LIN {X 0,Y 364.275,Z 621.196,A -85,B 0,C 180,E1 12256.474,E2 12256.474} C_VEL
LIN {X 0,Y 364.034,Z 587.813,A -85,B 0,C 180,E1 12257.54,E2 12257.54} C_VEL
LIN {X 0,Y 354.056,Z 549.53,A -85,B 0,C 180,E1 12259.048,E2 12259.048} C_VEL
LIN {X 0,Y 353.541,Z 549.53,A -85,B 0,C 180,E1 12266.307,E2 12266.307} C_VEL
LIN {X 0,Y 353.274,Z 549.53,A -85,B 0,C 180,E1 12273.738,E2 12273.738} C_VEL
LIN {X 0,Y 353.185,Z 549.53,A -85,B 0,C 180,E1 12279.866,E2 12279.866} C_VEL
LIN {X 0,Y 353.249,Z 549.563,A -85,B 0,C 180,E1 12286.159,E2 12286.159} C_VEL
LIN {X 0,Y 355.771,Z 555.279,A -85,B 0,C 180,E1 12286.913,E2 12286.913} C_VEL
LIN {X 0,Y 373.351,Z 588.547,A -85,B 0,C 180,E1 12291.308,E2 12291.308} C_VEL
LIN {X 0,Y 385.04,Z 618.639,A -85,B 0,C 180,E1 12294.556,E2 12294.556} C_VEL
LIN {X 0,Y 386.445,Z 626.078,A -85,B 0,C 180,E1 12295.26,E2 12295.26} C_VEL
LIN {X 0,Y 380.974,Z 661.138,A -85,B 0,C 180,E1 12297.839,E2 12297.839} C_VEL
LIN {X 0,Y 374.56,Z 693.358,A -85,B 0,C 180,E1 12301.251,E2 12301.251} C_VEL
LIN {X 0,Y 368.305,Z 721.793,A -85,B 0,C 180,E1 12305.491,E2 12305.491} C_VEL
LIN {X 0,Y 363.131,Z 744.325,A -85,B 0,C 180,E1 12310.113,E2 12310.113} C_VEL
LIN {X 0,Y 359.19,Z 762.864,A -85,B 0,C 180,E1 12315.399,E2 12315.399} C_VEL
LIN {X 0,Y 356.931,Z 776.042,A -85,B 0,C 180,E1 12320.877,E2 12320.877} C_VEL
LIN {X 0,Y 355.982,Z 784.021,A -85,B 0,C 180,E1 12326.354,E2 12326.354} C_VEL
LIN {X 0,Y 355.823,Z 786.74,A -85,B 0,C 180,E1 12330,E2 12330} C_VEL
LIN {X 0,Y 355.614,Z 787.304,A -85,B 0,C 180,E1 12334.869,E2 12334.869} C_VEL
LIN {X 0,Y 356.095,Z 782.784,A -85,B 0,C 180,E1 12340.995,E2 12340.995} C_VEL
LIN {X 0,Y 357.469,Z 773.674,A -85,B 0,C 180,E1 12346.558,E2 12346.558} C_VEL
LIN {X 0,Y 360.3,Z 759.136,A -85,B 0,C 180,E1 12352.147,E2 12352.147} C_VEL
LIN {X 0,Y 365.023,Z 739.076,A -85,B 0,C 180,E1 12357.433,E2 12357.433} C_VEL
LIN {X 0,Y 371.397,Z 713.51,A -85,B 0,C 180,E1 12362.225,E2 12362.225} C_VEL
LIN {X 0,Y 377.949,Z 685.061,A -85,B 0,C 180,E1 12366.085,E2 12366.085} C_VEL
LIN {X 0,Y 384.414,Z 652.218,A -85,B 0,C 180,E1 12369.256,E2 12369.256} C_VEL
LIN {X 0,Y 388.288,Z 623.748,A -85,B 0,C 180,E1 12371.277,E2 12371.277} C_VEL
LIN {X 0,Y 379.667,Z 599.13,A -85,B 0,C 180,E1 12374.088,E2 12374.088} C_VEL
LIN {X 0,Y 362.784,Z 566.88,A -85,B 0,C 180,E1 12378.529,E2 12378.529} C_VEL
LIN {X 0,Y 353.462,Z 550.572,A -85,B 0,C 180,E1 12381.288,E2 12381.288} C_VEL
LIN {X 0,Y 353.384,Z 549.53,A -85,B 0,C 180,E1 12381.533,E2 12381.533} C_VEL
LIN {X 0,Y 353.448,Z 549.53,A -85,B 0,C 180,E1 12389.174,E2 12389.174} C_VEL
LIN {X 0,Y 353.791,Z 549.53,A -85,B 0,C 180,E1 12394.746,E2 12394.746} C_VEL
LIN {X 0,Y 363.12,Z 590.42,A -85,B 0,C 180,E1 12396.235,E2 12396.235} C_VEL
LIN {X 0,Y 362.485,Z 640.026,A -85,B 0,C 180,E1 12397.587,E2 12397.587} C_VEL
LIN {X 0,Y 361.697,Z 666.836,A -85,B 0,C 180,E1 12399.26,E2 12399.26} C_VEL
LIN {X 0,Y 360.494,Z 691.605,A -85,B 0,C 180,E1 12401.855,E2 12401.855} C_VEL
LIN {X 0,Y 359.119,Z 711.774,A -85,B 0,C 180,E1 12405.143,E2 12405.143} C_VEL
LIN {X 0,Y 358.399,Z 725.013,A -85,B 0,C 180,E1 12408.458,E2 12408.458} C_VEL
LIN {X 0,Y 357.994,Z 734.312,A -85,B 0,C 180,E1 12412.298,E2 12412.298} C_VEL
LIN {X 0,Y 358.059,Z 737.826,A -85,B 0,C 180,E1 12415.159,E2 12415.159} C_VEL
LIN {X 0,Y 358.173,Z 738.62,A -85,B 0,C 180,E1 12417.58,E2 12417.58} C_VEL
LIN {X 0,Y 358.909,Z 736.002,A -85,B 0,C 180,E1 12421.199,E2 12421.199} C_VEL
LIN {X 0,Y 360.066,Z 728.623,A -85,B 0,C 180,E1 12424.803,E2 12424.803} C_VEL
LIN {X 0,Y 361.744,Z 715.298,A -85,B 0,C 180,E1 12428.39,E2 12428.39} C_VEL
LIN {X 0,Y 363.572,Z 696.667,A -85,B 0,C 180,E1 12431.517,E2 12431.517} C_VEL
LIN {X 0,Y 365.152,Z 674.086,A -85,B 0,C 180,E1 12433.913,E2 12433.913} C_VEL
LIN {X 0,Y 365.958,Z 647.126,A -85,B 0,C 180,E1 12435.618,E2 12435.618} C_VEL
LIN {X 0,Y 366.369,Z 584.89,A -85,B 0,C 180,E1 12437.501,E2 12437.501} C_VEL
LIN {X 0,Y 357.409,Z 558.523,A -85,B 0,C 180,E1 12439.203,E2 12439.203} C_VEL
LIN {X 0,Y 353.822,Z 549.53,A -85,B 0,C 180,E1 12439.944,E2 12439.944} C_VEL
LIN {X 0,Y 353.455,Z 549.53,A -85,B 0,C 180,E1 12446.277,E2 12446.277} C_VEL
LIN {X 0,Y 353.259,Z 549.53,A -85,B 0,C 180,E1 12454.23,E2 12454.23} C_VEL
LIN {X 0,Y 355.68,Z 555.181,A -85,B 0,C 180,E1 12455.037,E2 12455.037} C_VEL
LIN {X 0,Y 369.418,Z 576.894,A -85,B 0,C 180,E1 12458.683,E2 12458.683} C_VEL
LIN {X 0,Y 385.949,Z 608.362,A -85,B 0,C 180,E1 12462.881,E2 12462.881} C_VEL
LIN {X 0,Y 391.213,Z 623.866,A -85,B 0,C 180,E1 12464.463,E2 12464.463} C_VEL
LIN {X 0,Y 395.036,Z 639.941,A -85,B 0,C 180,E1 12465.933,E2 12465.933} C_VEL
LIN {X 0,Y 388.164,Z 682.729,A -85,B 0,C 180,E1 12468.377,E2 12468.377} C_VEL
LIN {X 0,Y 380.662,Z 723.232,A -85,B 0,C 180,E1 12471.698,E2 12471.698} C_VEL
LIN {X 0,Y 373.751,Z 755.378,A -85,B 0,C 180,E1 12475.4,E2 12475.4} C_VEL
LIN {X 0,Y 367.102,Z 783.844,A -85,B 0,C 180,E1 12479.95,E2 12479.95} C_VEL
LIN {X 0,Y 361.472,Z 808.192,A -85,B 0,C 180,E1 12485.322,E2 12485.322} C_VEL
LIN {X 0,Y 357.553,Z 827.685,A -85,B 0,C 180,E1 12491.408,E2 12491.408} C_VEL
LIN {X 0,Y 355.887,Z 840.326,A -85,B 0,C 180,E1 12497.199,E2 12497.199} C_VEL
LIN {X 0,Y 355.241,Z 848.253,A -85,B 0,C 180,E1 12503.285,E2 12503.285} C_VEL
LIN {X 0,Y 355.256,Z 851.147,A -85,B 0,C 180,E1 12508.729,E2 12508.729} C_VEL
LIN {X 0,Y 352.765,Z 851.098,A -85,B 0,C 180,E1 12510.813,E2 12510.813} C_VEL
LIN {X 0,Y 347.396,Z 849.644,A -85,B 0,C 180,E1 12513.951,E2 12513.951} C_VEL
LIN {X 0,Y 347.31,Z 849.375,A -85,B 0,C 180,E1 12514.316,E2 12514.316} C_VEL
LIN {X 0,Y 347.573,Z 844.231,A -85,B 0,C 180,E1 12520.002,E2 12520.002} C_VEL
LIN {X 0,Y 348.862,Z 833.205,A -85,B 0,C 180,E1 12526.331,E2 12526.331} C_VEL
LIN {X 0,Y 351.743,Z 816.942,A -85,B 0,C 180,E1 12532.382,E2 12532.382} C_VEL
LIN {X 0,Y 356.706,Z 794.96,A -85,B 0,C 180,E1 12538.078,E2 12538.078} C_VEL
LIN {X 0,Y 362.874,Z 769.059,A -85,B 0,C 180,E1 12542.937,E2 12542.937} C_VEL
LIN {X 0,Y 369.91,Z 738.065,A -85,B 0,C 180,E1 12547.128,E2 12547.128} C_VEL
LIN {X 0,Y 377.086,Z 701.811,A -85,B 0,C 180,E1 12550.606,E2 12550.606} C_VEL
LIN {X 0,Y 384.419,Z 658.93,A -85,B 0,C 180,E1 12553.528,E2 12553.528} C_VEL
LIN {X 0,Y 387.166,Z 639.433,A -85,B 0,C 180,E1 12554.558,E2 12554.558} C_VEL
LIN {X 0,Y 379.222,Z 613.621,A -85,B 0,C 180,E1 12557.069,E2 12557.069} C_VEL
LIN {X 0,Y 363.452,Z 581.4,A -85,B 0,C 180,E1 12561.01,E2 12561.01} C_VEL
LIN {X 0,Y 347.32,Z 554.675,A -85,B 0,C 180,E1 12565.104,E2 12565.104} C_VEL
LIN {X 0,Y 345.809,Z 552.078,A -85,B 0,C 180,E1 12565.608,E2 12565.608} C_VEL
LIN {X 0,Y 353.795,Z 566.714,A -85,B 0,C 180,E1 12567.716,E2 12567.716} C_VEL
LIN {X 0,Y 361.627,Z 587.377,A -85,B 0,C 180,E1 12569.616,E2 12569.616} C_VEL
LIN {X 0,Y 362.821,Z 598.343,A -85,B 0,C 180,E1 12570.16,E2 12570.16} C_VEL
LIN {X 0,Y 361.897,Z 640.267,A -85,B 0,C 180,E1 12571.732,E2 12571.732} C_VEL
LIN {X 0,Y 360.473,Z 667.942,A -85,B 0,C 180,E1 12573.669,E2 12573.669} C_VEL
LIN {X 0,Y 358.319,Z 692.777,A -85,B 0,C 180,E1 12576.423,E2 12576.423} C_VEL
LIN {X 0,Y 355.91,Z 713.04,A -85,B 0,C 180,E1 12579.869,E2 12579.869} C_VEL
LIN {X 0,Y 353.542,Z 727.584,A -85,B 0,C 180,E1 12583.724,E2 12583.724} C_VEL
LIN {X 0,Y 351.936,Z 736.22,A -85,B 0,C 180,E1 12587.626,E2 12587.626} C_VEL
LIN {X 0,Y 350.714,Z 740.148,A -85,B 0,C 180,E1 12591.777,E2 12591.777} C_VEL
LIN {X 0,Y 350.188,Z 738.761,A -85,B 0,C 180,E1 12596.3,E2 12596.3} C_VEL
LIN {X 0,Y 350.267,Z 731.975,A -85,B 0,C 180,E1 12600.623,E2 12600.623} C_VEL
LIN {X 0,Y 350.905,Z 719.455,A -85,B 0,C 180,E1 12604.94,E2 12604.94} C_VEL
LIN {X 0,Y 352.138,Z 701.16,A -85,B 0,C 180,E1 12608.942,E2 12608.942} C_VEL
LIN {X 0,Y 353.808,Z 678.257,A -85,B 0,C 180,E1 12612.319,E2 12612.319} C_VEL
LIN {X 0,Y 355.433,Z 652.196,A -85,B 0,C 180,E1 12614.911,E2 12614.911} C_VEL
LIN {X 0,Y 356.666,Z 622.078,A -85,B 0,C 180,E1 12616.775,E2 12616.775} C_VEL
LIN {X 0,Y 356.435,Z 589.165,A -85,B 0,C 180,E1 12617.849,E2 12617.849} C_VEL
LIN {X 0,Y 346.097,Z 549.53,A -85,B 0,C 180,E1 12619.504,E2 12619.504} C_VEL
LIN {X 0,Y 345.69,Z 549.53,A -85,B 0,C 180,E1 12625.889,E2 12625.889} C_VEL
LIN {X 0,Y 345.366,Z 549.53,A -85,B 0,C 180,E1 12633.875,E2 12633.875} C_VEL
LIN {X 0,Y 345.147,Z 549.53,A -85,B 0,C 180,E1 12640.989,E2 12640.989} C_VEL
LIN {X 0,Y 345.396,Z 550.336,A -85,B 0,C 180,E1 12644.716,E2 12644.716} C_VEL
LIN {X 0,Y 365.498,Z 588.003,A -85,B 0,C 180,E1 12650.154,E2 12650.154} C_VEL
LIN {X 0,Y 377.255,Z 616.784,A -85,B 0,C 180,E1 12653.451,E2 12653.451} C_VEL
LIN {X 0,Y 379.873,Z 629.008,A -85,B 0,C 180,E1 12654.681,E2 12654.681} C_VEL
LIN {X 0,Y 374.08,Z 663.933,A -85,B 0,C 180,E1 12657.344,E2 12657.344} C_VEL
LIN {X 0,Y 367.466,Z 695.539,A -85,B 0,C 180,E1 12660.811,E2 12660.811} C_VEL
LIN {X 0,Y 360.795,Z 724.424,A -85,B 0,C 180,E1 12665.274,E2 12665.274} C_VEL
LIN {X 0,Y 355.017,Z 748.245,A -85,B 0,C 180,E1 12670.442,E2 12670.442} C_VEL
LIN {X 0,Y 351.235,Z 765.466,A -85,B 0,C 180,E1 12675.697,E2 12675.697} C_VEL
LIN {X 0,Y 349.003,Z 777.905,A -85,B 0,C 180,E1 12681.295,E2 12681.295} C_VEL
LIN {X 0,Y 348.067,Z 785.91,A -85,B 0,C 180,E1 12687.515,E2 12687.515} C_VEL
LIN {X 0,Y 347.697,Z 788.224,A -85,B 0,C 180,E1 12693.328,E2 12693.328} C_VEL
LIN {X 0,Y 347.921,Z 785.975,A -85,B 0,C 180,E1 12698.733,E2 12698.733} C_VEL
LIN {X 0,Y 348.944,Z 779.227,A -85,B 0,C 180,E1 12704.263,E2 12704.263} C_VEL
LIN {X 0,Y 351.414,Z 766.905,A -85,B 0,C 180,E1 12710.095,E2 12710.095} C_VEL
LIN {X 0,Y 355.623,Z 748.992,A -85,B 0,C 180,E1 12715.74,E2 12715.74} C_VEL
LIN {X 0,Y 361.44,Z 726.447,A -85,B 0,C 180,E1 12720.735,E2 12720.735} C_VEL
LIN {X 0,Y 368.414,Z 698.59,A -85,B 0,C 180,E1 12725.174,E2 12725.174} C_VEL
LIN {X 0,Y 375.267,Z 667.967,A -85,B 0,C 180,E1 12728.674,E2 12728.674} C_VEL
LIN {X 0,Y 381.53,Z 633.671,A -85,B 0,C 180,E1 12731.384,E2 12731.384} C_VEL
LIN {X 0,Y 381.832,Z 625.306,A -85,B 0,C 180,E1 12732.03,E2 12732.03} C_VEL
LIN {X 0,Y 372.912,Z 600.763,A -85,B 0,C 180,E1 12735.01,E2 12735.01} C_VEL
LIN {X 0,Y 357.776,Z 571.815,A -85,B 0,C 180,E1 12739.191,E2 12739.191} C_VEL
LIN {X 0,Y 347.598,Z 554.926,A -85,B 0,C 180,E1 12742.297,E2 12742.297} C_VEL
LIN {X 0,Y 345.489,Z 549.53,A -85,B 0,C 180,E1 12743.254,E2 12743.254} C_VEL
LIN {X 0,Y 345.502,Z 549.53,A -85,B 0,C 180,E1 12750.883,E2 12750.883} C_VEL
LIN {X 0,Y 345.858,Z 550.002,A -85,B 0,C 180,E1 12754.381,E2 12754.381} C_VEL
LIN {X 0,Y 355.487,Z 591.258,A -85,B 0,C 180,E1 12755.919,E2 12755.919} C_VEL
LIN {X 0,Y 354.851,Z 640.437,A -85,B 0,C 180,E1 12757.285,E2 12757.285} C_VEL
LIN {X 0,Y 353.992,Z 668.172,A -85,B 0,C 180,E1 12759.043,E2 12759.043} C_VEL
LIN {X 0,Y 352.778,Z 692.243,A -85,B 0,C 180,E1 12761.605,E2 12761.605} C_VEL
LIN {X 0,Y 351.399,Z 711.894,A -85,B 0,C 180,E1 12764.809,E2 12764.809} C_VEL
LIN {X 0,Y 350.639,Z 725.614,A -85,B 0,C 180,E1 12768.199,E2 12768.199} C_VEL
LIN {X 0,Y 350.203,Z 735.78,A -85,B 0,C 180,E1 12772.384,E2 12772.384} C_VEL
LIN {X 0,Y 350.286,Z 739.04,A -85,B 0,C 180,E1 12775.052,E2 12775.052} C_VEL
LIN {X 0,Y 350.404,Z 740.035,A -85,B 0,C 180,E1 12777.526,E2 12777.526} C_VEL
LIN {X 0,Y 351.187,Z 737.683,A -85,B 0,C 180,E1 12781.225,E2 12781.225} C_VEL
LIN {X 0,Y 352.424,Z 730.53,A -85,B 0,C 180,E1 12784.907,E2 12784.907} C_VEL
LIN {X 0,Y 354.226,Z 717.584,A -85,B 0,C 180,E1 12788.569,E2 12788.569} C_VEL
LIN {X 0,Y 356.159,Z 699.356,A -85,B 0,C 180,E1 12791.76,E2 12791.76} C_VEL
LIN {X 0,Y 357.859,Z 677.477,A -85,B 0,C 180,E1 12794.214,E2 12794.214} C_VEL
LIN {X 0,Y 358.796,Z 652.243,A -85,B 0,C 180,E1 12795.938,E2 12795.938} C_VEL
LIN {X 0,Y 359.596,Z 602.628,A -85,B 0,C 180,E1 12797.543,E2 12797.543} C_VEL
LIN {X 0,Y 359.362,Z 586.315,A -85,B 0,C 180,E1 12798.081,E2 12798.081} C_VEL
LIN {X 0,Y 351.153,Z 562.179,A -85,B 0,C 180,E1 12799.754,E2 12799.754} C_VEL
LIN {X 0,Y 345.822,Z 549.53,A -85,B 0,C 180,E1 12800.927,E2 12800.927} C_VEL
LIN {X 0,Y 345.407,Z 549.53,A -85,B 0,C 180,E1 12808.716,E2 12808.716} C_VEL
LIN {X 0,Y 345.358,Z 550.3,A -85,B 0,C 180,E1 12812.478,E2 12812.478} C_VEL
LIN {X 0,Y 348.222,Z 555.583,A -85,B 0,C 180,E1 12813.406,E2 12813.406} C_VEL
LIN {X 0,Y 364.524,Z 581.656,A -85,B 0,C 180,E1 12818.041,E2 12818.041} C_VEL
LIN {X 0,Y 380.588,Z 613.052,A -85,B 0,C 180,E1 12822.373,E2 12822.373} C_VEL
LIN {X 0,Y 385.375,Z 627.724,A -85,B 0,C 180,E1 12823.926,E2 12823.926} C_VEL
LIN {X 0,Y 388.533,Z 642.853,A -85,B 0,C 180,E1 12825.323,E2 12825.323} C_VEL
LIN {X 0,Y 381.588,Z 683.907,A -85,B 0,C 180,E1 12827.751,E2 12827.751} C_VEL
LIN {X 0,Y 373.888,Z 723.78,A -85,B 0,C 180,E1 12831.084,E2 12831.084} C_VEL
LIN {X 0,Y 366.711,Z 755.537,A -85,B 0,C 180,E1 12834.818,E2 12834.818} C_VEL
LIN {X 0,Y 359.692,Z 784.163,A -85,B 0,C 180,E1 12839.517,E2 12839.517} C_VEL
LIN {X 0,Y 354.031,Z 807.428,A -85,B 0,C 180,E1 12844.768,E2 12844.768} C_VEL
LIN {X 0,Y 349.891,Z 826.728,A -85,B 0,C 180,E1 12850.895,E2 12850.895} C_VEL
LIN {X 0,Y 348.024,Z 839.624,A -85,B 0,C 180,E1 12856.905,E2 12856.905} C_VEL
LIN {X 0,Y 347.449,Z 847.066,A -85,B 0,C 180,E1 12862.512,E2 12862.512} C_VEL
LIN {X 0,Y 347.394,Z 850.449,A -85,B 0,C 180,E1 12868.746,E2 12868.746} C_VEL
LIN {X 0,Y 347.31,Z 849.375,A -85,B 0,C 180,E1 12874.316,E2 12874.316} C_VEL
LIN {X 0,Y 344.863,Z 847.822,A -85,B 0,C 180,E1 12876.434,E2 12876.434} C_VEL
LIN {X 0,Y 339.68,Z 843.795,A -85,B 0,C 180,E1 12879.971,E2 12879.971} C_VEL
LIN {X 0,Y 340.91,Z 833.804,A -85,B 0,C 180,E1 12886.062,E2 12886.062} C_VEL
LIN {X 0,Y 343.839,Z 817.537,A -85,B 0,C 180,E1 12892.415,E2 12892.415} C_VEL
LIN {X 0,Y 348.804,Z 796.429,A -85,B 0,C 180,E1 12898.159,E2 12898.159} C_VEL
LIN {X 0,Y 355.392,Z 769.991,A -85,B 0,C 180,E1 12903.307,E2 12903.307} C_VEL
LIN {X 0,Y 362.653,Z 739.67,A -85,B 0,C 180,E1 12907.56,E2 12907.56} C_VEL
LIN {X 0,Y 370,Z 704.126,A -85,B 0,C 180,E1 12911.084,E2 12911.084} C_VEL
LIN {X 0,Y 377.831,Z 660.691,A -85,B 0,C 180,E1 12914.144,E2 12914.144} C_VEL
LIN {X 0,Y 380.362,Z 640.833,A -85,B 0,C 180,E1 12915.269,E2 12915.269} C_VEL
LIN {X 0,Y 373.295,Z 617.367,A -85,B 0,C 180,E1 12917.646,E2 12917.646} C_VEL
LIN {X 0,Y 358.128,Z 585.709,A -85,B 0,C 180,E1 12921.676,E2 12921.676} C_VEL
LIN {X 0,Y 343.338,Z 561.006,A -85,B 0,C 180,E1 12925.614,E2 12925.614} C_VEL
LIN {X 0,Y 351.87,Z 579.207,A -85,B 0,C 180,E1 12927.997,E2 12927.997} C_VEL
LIN {X 0,Y 356.525,Z 595.345,A -85,B 0,C 180,E1 12929.306,E2 12929.306} C_VEL
LIN {X 0,Y 355.248,Z 641.4,A -85,B 0,C 180,E1 12931.076,E2 12931.076} C_VEL
LIN {X 0,Y 353.657,Z 669.446,A -85,B 0,C 180,E1 12933.079,E2 12933.079} C_VEL
LIN {X 0,Y 351.284,Z 694.52,A -85,B 0,C 180,E1 12935.921,E2 12935.921} C_VEL
LIN {X 0,Y 348.662,Z 714.712,A -85,B 0,C 180,E1 12939.432,E2 12939.432} C_VEL
LIN {X 0,Y 346.196,Z 728.782,A -85,B 0,C 180,E1 12943.206,E2 12943.206} C_VEL
LIN {X 0,Y 344.35,Z 737.82,A -85,B 0,C 180,E1 12947.349,E2 12947.349} C_VEL
LIN {X 0,Y 343.5,Z 740.75,A -85,B 0,C 180,E1 12949.885,E2 12949.885} C_VEL
LIN {X 0,Y 342.837,Z 741.814,A -85,B 0,C 180,E1 12952.418,E2 12952.418} C_VEL
LIN {X 0,Y 342.421,Z 740.159,A -85,B 0,C 180,E1 12956.216,E2 12956.216} C_VEL
LIN {X 0,Y 342.462,Z 733.251,A -85,B 0,C 180,E1 12960.637,E2 12960.637} C_VEL
LIN {X 0,Y 343.106,Z 720.542,A -85,B 0,C 180,E1 12965.052,E2 12965.052} C_VEL
LIN {X 0,Y 344.395,Z 702.255,A -85,B 0,C 180,E1 12969.097,E2 12969.097} C_VEL
LIN {X 0,Y 346.119,Z 678.748,A -85,B 0,C 180,E1 12972.597,E2 12972.597} C_VEL
LIN {X 0,Y 347.838,Z 651.106,A -85,B 0,C 180,E1 12975.335,E2 12975.335} C_VEL
LIN {X 0,Y 349.067,Z 621.464,A -85,B 0,C 180,E1 12977.149,E2 12977.149} C_VEL
LIN {X 0,Y 348.829,Z 590.551,A -85,B 0,C 180,E1 12978.168,E2 12978.168} C_VEL
LIN {X 0,Y 338.109,Z 549.53,A -85,B 0,C 180,E1 12979.9,E2 12979.9} C_VEL
LIN {X 0,Y 337.654,Z 549.53,A -85,B 0,C 180,E1 12986.631,E2 12986.631} C_VEL
LIN {X 0,Y 337.456,Z 549.53,A -85,B 0,C 180,E1 12992.46,E2 12992.46} C_VEL
LIN {X 0,Y 337.191,Z 549.53,A -85,B 0,C 180,E1 13000.459,E2 13000.459} C_VEL
LIN {X 0,Y 337.244,Z 549.687,A -85,B 0,C 180,E1 13003.006,E2 13003.006} C_VEL
LIN {X 0,Y 339.887,Z 555.337,A -85,B 0,C 180,E1 13003.897,E2 13003.897} C_VEL
LIN {X 0,Y 356.219,Z 584.601,A -85,B 0,C 180,E1 13008.537,E2 13008.537} C_VEL
LIN {X 0,Y 369.084,Z 614.096,A -85,B 0,C 180,E1 13012.169,E2 13012.169} C_VEL
LIN {X 0,Y 373.502,Z 630.833,A -85,B 0,C 180,E1 13014.018,E2 13014.018} C_VEL
LIN {X 0,Y 367.55,Z 665.137,A -85,B 0,C 180,E1 13016.689,E2 13016.689} C_VEL
LIN {X 0,Y 360.4,Z 697.715,A -85,B 0,C 180,E1 13020.354,E2 13020.354} C_VEL
LIN {X 0,Y 353.665,Z 725.396,A -85,B 0,C 180,E1 13024.741,E2 13024.741} C_VEL
LIN {X 0,Y 347.612,Z 749.134,A -85,B 0,C 180,E1 13030.008,E2 13030.008} C_VEL
LIN {X 0,Y 343.615,Z 766.17,A -85,B 0,C 180,E1 13035.319,E2 13035.319} C_VEL
LIN {X 0,Y 341.209,Z 778.693,A -85,B 0,C 180,E1 13041.095,E2 13041.095} C_VEL
LIN {X 0,Y 340.223,Z 786.654,A -85,B 0,C 180,E1 13047.458,E2 13047.458} C_VEL
LIN {X 0,Y 339.893,Z 788.872,A -85,B 0,C 180,E1 13052.545,E2 13052.545} C_VEL
LIN {X 0,Y 339.984,Z 787.519,A -85,B 0,C 180,E1 13057.653,E2 13057.653} C_VEL
LIN {X 0,Y 340.82,Z 782.156,A -85,B 0,C 180,E1 13063.048,E2 13063.048} C_VEL
LIN {X 0,Y 343.109,Z 770.855,A -85,B 0,C 180,E1 13069.205,E2 13069.205} C_VEL
LIN {X 0,Y 347.265,Z 753.859,A -85,B 0,C 180,E1 13075.115,E2 13075.115} C_VEL
LIN {X 0,Y 353.262,Z 731.665,A -85,B 0,C 180,E1 13080.486,E2 13080.486} C_VEL
LIN {X 0,Y 360.312,Z 705.295,A -85,B 0,C 180,E1 13085.028,E2 13085.028} C_VEL
LIN {X 0,Y 367.7,Z 674.772,A -85,B 0,C 180,E1 13088.798,E2 13088.798} C_VEL
LIN {X 0,Y 374.409,Z 641.452,A -85,B 0,C 180,E1 13091.677,E2 13091.677} C_VEL
LIN {X 0,Y 375.885,Z 629.111,A -85,B 0,C 180,E1 13092.566,E2 13092.566} C_VEL
LIN {X 0,Y 366.781,Z 603.545,A -85,B 0,C 180,E1 13095.818,E2 13095.818} C_VEL
LIN {X 0,Y 351.189,Z 573.486,A -85,B 0,C 180,E1 13100.383,E2 13100.383} C_VEL
LIN {X 0,Y 339.956,Z 555.177,A -85,B 0,C 180,E1 13104.066,E2 13104.066} C_VEL
LIN {X 0,Y 337.616,Z 549.53,A -85,B 0,C 180,E1 13105.266,E2 13105.266} C_VEL
LIN {X 0,Y 337.882,Z 549.794,A -85,B 0,C 180,E1 13113.965,E2 13113.965} C_VEL
LIN {X 0,Y 347.872,Z 591.849,A -85,B 0,C 180,E1 13115.597,E2 13115.597} C_VEL
LIN {X 0,Y 347.197,Z 642.226,A -85,B 0,C 180,E1 13117.051,E2 13117.051} C_VEL
LIN {X 0,Y 346.312,Z 668.669,A -85,B 0,C 180,E1 13118.758,E2 13118.758} C_VEL
LIN {X 0,Y 345.075,Z 692.964,A -85,B 0,C 180,E1 13121.365,E2 13121.365} C_VEL
LIN {X 0,Y 343.604,Z 713.242,A -85,B 0,C 180,E1 13124.716,E2 13124.716} C_VEL
LIN {X 0,Y 342.768,Z 728.188,A -85,B 0,C 180,E1 13128.568,E2 13128.568} C_VEL
LIN {X 0,Y 342.39,Z 737.074,A -85,B 0,C 180,E1 13132.396,E2 13132.396} C_VEL
LIN {X 0,Y 342.482,Z 740.255,A -85,B 0,C 180,E1 13134.939,E2 13134.939} C_VEL
LIN {X 0,Y 342.63,Z 741.426,A -85,B 0,C 180,E1 13137.47,E2 13137.47} C_VEL
LIN {X 0,Y 343.462,Z 739.36,A -85,B 0,C 180,E1 13141.253,E2 13141.253} C_VEL
LIN {X 0,Y 344.79,Z 732.504,A -85,B 0,C 180,E1 13145.016,E2 13145.016} C_VEL
LIN {X 0,Y 346.703,Z 719.887,A -85,B 0,C 180,E1 13148.757,E2 13148.757} C_VEL
LIN {X 0,Y 348.849,Z 702.179,A -85,B 0,C 180,E1 13152.01,E2 13152.01} C_VEL
LIN {X 0,Y 350.643,Z 680.162,A -85,B 0,C 180,E1 13154.595,E2 13154.595} C_VEL
LIN {X 0,Y 351.748,Z 654.629,A -85,B 0,C 180,E1 13156.426,E2 13156.426} C_VEL
LIN {X 0,Y 352.598,Z 606.377,A -85,B 0,C 180,E1 13158.072,E2 13158.072} C_VEL
LIN {X 0,Y 352.523,Z 587.855,A -85,B 0,C 180,E1 13158.704,E2 13158.704} C_VEL
LIN {X 0,Y 344.339,Z 564.234,A -85,B 0,C 180,E1 13160.471,E2 13160.471} C_VEL
LIN {X 0,Y 337.887,Z 549.53,A -85,B 0,C 180,E1 13161.96,E2 13161.96} C_VEL
LIN {X 0,Y 337.423,Z 549.53,A -85,B 0,C 180,E1 13169.843,E2 13169.843} C_VEL
LIN {X 0,Y 337.438,Z 550.022,A -85,B 0,C 180,E1 13170.459,E2 13170.459} C_VEL
LIN {X 0,Y 339.896,Z 555.205,A -85,B 0,C 180,E1 13171.373,E2 13171.373} C_VEL
LIN {X 0,Y 353.957,Z 576.827,A -85,B 0,C 180,E1 13175.75,E2 13175.75} C_VEL
LIN {X 0,Y 370.434,Z 607.264,A -85,B 0,C 180,E1 13180.477,E2 13180.477} C_VEL
LIN {X 0,Y 378.796,Z 627.97,A -85,B 0,C 180,E1 13183.032,E2 13183.032} C_VEL
LIN {X 0,Y 382.126,Z 645.572,A -85,B 0,C 180,E1 13184.691,E2 13184.691} C_VEL
LIN {X 0,Y 374.746,Z 686.869,A -85,B 0,C 180,E1 13187.228,E2 13187.228} C_VEL
LIN {X 0,Y 366.874,Z 725.637,A -85,B 0,C 180,E1 13190.576,E2 13190.576} C_VEL
LIN {X 0,Y 359.481,Z 756.528,A -85,B 0,C 180,E1 13194.341,E2 13194.341} C_VEL
LIN {X 0,Y 352.319,Z 784.494,A -85,B 0,C 180,E1 13199.067,E2 13199.067} C_VEL
LIN {X 0,Y 346.317,Z 807.804,A -85,B 0,C 180,E1 13204.511,E2 13204.511} C_VEL
LIN {X 0,Y 342.074,Z 826.59,A -85,B 0,C 180,E1 13210.677,E2 13210.677} C_VEL
LIN {X 0,Y 340.085,Z 839.842,A -85,B 0,C 180,E1 13217.18,E2 13217.18} C_VEL
LIN {X 0,Y 339.568,Z 846.367,A -85,B 0,C 180,E1 13222.337,E2 13222.337} C_VEL
LIN {X 0,Y 339.515,Z 849.531,A -85,B 0,C 180,E1 13227.452,E2 13227.452} C_VEL
LIN {X 0,Y 339.584,Z 849.534,A -85,B 0,C 180,E1 13232.547,E2 13232.547} C_VEL
LIN {X 0,Y 339.65,Z 845.012,A -85,B 0,C 180,E1 13238.946,E2 13238.946} C_VEL
LIN {X 0,Y 339.68,Z 843.795,A -85,B 0,C 180,E1 13239.971,E2 13239.971} C_VEL
LIN {X 0,Y 337.432,Z 840.822,A -85,B 0,C 180,E1 13242.104,E2 13242.104} C_VEL
LIN {X 0,Y 332.839,Z 835.253,A -85,B 0,C 180,E1 13245.277,E2 13245.277} C_VEL
LIN {X 0,Y 332.854,Z 834.556,A -85,B 0,C 180,E1 13245.638,E2 13245.638} C_VEL
LIN {X 0,Y 335.772,Z 818.735,A -85,B 0,C 180,E1 13252.255,E2 13252.255} C_VEL
LIN {X 0,Y 340.763,Z 798.388,A -85,B 0,C 180,E1 13258.092,E2 13258.092} C_VEL
LIN {X 0,Y 347.286,Z 773.377,A -85,B 0,C 180,E1 13263.273,E2 13263.273} C_VEL
LIN {X 0,Y 354.65,Z 744.116,A -85,B 0,C 180,E1 13267.652,E2 13267.652} C_VEL
LIN {X 0,Y 362.234,Z 710.101,A -85,B 0,C 180,E1 13271.261,E2 13271.261} C_VEL
LIN {X 0,Y 370.472,Z 667.073,A -85,B 0,C 180,E1 13274.496,E2 13274.496} C_VEL
LIN {X 0,Y 373.913,Z 643.392,A -85,B 0,C 180,E1 13275.887,E2 13275.887} C_VEL
LIN {X 0,Y 367.627,Z 621.743,A -85,B 0,C 180,E1 13278.168,E2 13278.168} C_VEL
LIN {X 0,Y 352.328,Z 588.924,A -85,B 0,C 180,E1 13282.49,E2 13282.49} C_VEL
LIN {X 0,Y 341.03,Z 570.39,A -85,B 0,C 180,E1 13285.61,E2 13285.61} C_VEL
LIN {X 0,Y 347.694,Z 587.158,A -85,B 0,C 180,E1 13287.737,E2 13287.737} C_VEL
LIN {X 0,Y 350.227,Z 599.073,A -85,B 0,C 180,E1 13288.631,E2 13288.631} C_VEL
LIN {X 0,Y 348.648,Z 644.316,A -85,B 0,C 180,E1 13290.477,E2 13290.477} C_VEL
LIN {X 0,Y 346.788,Z 673.069,A -85,B 0,C 180,E1 13292.644,E2 13292.644} C_VEL
LIN {X 0,Y 344.169,Z 697.583,A -85,B 0,C 180,E1 13295.563,E2 13295.563} C_VEL
LIN {X 0,Y 341.442,Z 716.782,A -85,B 0,C 180,E1 13299.035,E2 13299.035} C_VEL
LIN {X 0,Y 338.959,Z 729.807,A -85,B 0,C 180,E1 13302.589,E2 13302.589} C_VEL
LIN {X 0,Y 336.793,Z 739.434,A -85,B 0,C 180,E1 13307.06,E2 13307.06} C_VEL
LIN {X 0,Y 335.86,Z 742.315,A -85,B 0,C 180,E1 13309.652,E2 13309.652} C_VEL
LIN {X 0,Y 335.133,Z 743.319,A -85,B 0,C 180,E1 13312.243,E2 13312.243} C_VEL
LIN {X 0,Y 334.653,Z 741.555,A -85,B 0,C 180,E1 13316.128,E2 13316.128} C_VEL
LIN {X 0,Y 334.671,Z 734.48,A -85,B 0,C 180,E1 13320.652,E2 13320.652} C_VEL
LIN {X 0,Y 335.314,Z 721.58,A -85,B 0,C 180,E1 13325.17,E2 13325.17} C_VEL
LIN {X 0,Y 336.681,Z 702.724,A -85,B 0,C 180,E1 13329.379,E2 13329.379} C_VEL
LIN {X 0,Y 338.457,Z 679.243,A -85,B 0,C 180,E1 13332.887,E2 13332.887} C_VEL
LIN {X 0,Y 340.158,Z 652.359,A -85,B 0,C 180,E1 13335.585,E2 13335.585} C_VEL
LIN {X 0,Y 341.431,Z 622.478,A -85,B 0,C 180,E1 13337.45,E2 13337.45} C_VEL
LIN {X 0,Y 341.148,Z 591.395,A -85,B 0,C 180,E1 13338.506,E2 13338.506} C_VEL
LIN {X 0,Y 330.183,Z 549.53,A -85,B 0,C 180,E1 13340.348,E2 13340.348} C_VEL
LIN {X 0,Y 329.681,Z 549.53,A -85,B 0,C 180,E1 13347.247,E2 13347.247} C_VEL
LIN {X 0,Y 329.325,Z 549.53,A -85,B 0,C 180,E1 13354.425,E2 13354.425} C_VEL
LIN {X 0,Y 329.318,Z 550.196,A -85,B 0,C 180,E1 13361.257,E2 13361.257} C_VEL
LIN {X 0,Y 332.287,Z 555.687,A -85,B 0,C 180,E1 13362.292,E2 13362.292} C_VEL
LIN {X 0,Y 348.61,Z 584.636,A -85,B 0,C 180,E1 13367.261,E2 13367.261} C_VEL
LIN {X 0,Y 362.016,Z 614.646,A -85,B 0,C 180,E1 13371.194,E2 13371.194} C_VEL
LIN {X 0,Y 367.194,Z 632.594,A -85,B 0,C 180,E1 13373.327,E2 13373.327} C_VEL
LIN {X 0,Y 360.74,Z 667.922,A -85,B 0,C 180,E1 13376.156,E2 13376.156} C_VEL
LIN {X 0,Y 353.364,Z 699.882,A -85,B 0,C 180,E1 13379.879,E2 13379.879} C_VEL
LIN {X 0,Y 346.159,Z 727.939,A -85,B 0,C 180,E1 13384.499,E2 13384.499} C_VEL
LIN {X 0,Y 339.91,Z 751.238,A -85,B 0,C 180,E1 13389.874,E2 13389.874} C_VEL
LIN {X 0,Y 335.426,Z 769.475,A -85,B 0,C 180,E1 13395.978,E2 13395.978} C_VEL
LIN {X 0,Y 333.083,Z 781.567,A -85,B 0,C 180,E1 13402.188,E2 13402.188} C_VEL
LIN {X 0,Y 332.363,Z 787.4,A -85,B 0,C 180,E1 13407.398,E2 13407.398} C_VEL
LIN {X 0,Y 332.048,Z 789.583,A -85,B 0,C 180,E1 13412.606,E2 13412.606} C_VEL
LIN {X 0,Y 332.156,Z 788.2,A -85,B 0,C 180,E1 13417.835,E2 13417.835} C_VEL
LIN {X 0,Y 333.344,Z 781.35,A -85,B 0,C 180,E1 13424.419,E2 13424.419} C_VEL
LIN {X 0,Y 335.991,Z 769.578,A -85,B 0,C 180,E1 13430.452,E2 13430.452} C_VEL
LIN {X 0,Y 340.562,Z 752.376,A -85,B 0,C 180,E1 13436.305,E2 13436.305} C_VEL
LIN {X 0,Y 346.826,Z 730.617,A -85,B 0,C 180,E1 13441.478,E2 13441.478} C_VEL
LIN {X 0,Y 354.266,Z 703.996,A -85,B 0,C 180,E1 13446.05,E2 13446.05} C_VEL
LIN {X 0,Y 362.028,Z 672.858,A -85,B 0,C 180,E1 13449.839,E2 13449.839} C_VEL
LIN {X 0,Y 369.121,Z 638.224,A -85,B 0,C 180,E1 13452.742,E2 13452.742} C_VEL
LIN {X 0,Y 369.437,Z 630.469,A -85,B 0,C 180,E1 13453.4,E2 13453.4} C_VEL
LIN {X 0,Y 359.697,Z 603.953,A -85,B 0,C 180,E1 13456.97,E2 13456.97} C_VEL
LIN {X 0,Y 343.883,Z 574.042,A -85,B 0,C 180,E1 13461.897,E2 13461.897} C_VEL
LIN {X 0,Y 332.139,Z 555.211,A -85,B 0,C 180,E1 13466.067,E2 13466.067} C_VEL
LIN {X 0,Y 329.695,Z 549.53,A -85,B 0,C 180,E1 13467.379,E2 13467.379} C_VEL
LIN {X 0,Y 329.872,Z 549.53,A -85,B 0,C 180,E1 13473.519,E2 13473.519} C_VEL
LIN {X 0,Y 340.237,Z 593.097,A -85,B 0,C 180,E1 13475.281,E2 13475.281} C_VEL
LIN {X 0,Y 339.524,Z 643.103,A -85,B 0,C 180,E1 13476.762,E2 13476.762} C_VEL
LIN {X 0,Y 338.59,Z 670.681,A -85,B 0,C 180,E1 13478.592,E2 13478.592} C_VEL
LIN {X 0,Y 337.312,Z 694.307,A -85,B 0,C 180,E1 13481.199,E2 13481.199} C_VEL
LIN {X 0,Y 335.837,Z 714.334,A -85,B 0,C 180,E1 13484.576,E2 13484.576} C_VEL
LIN {X 0,Y 335.007,Z 728.743,A -85,B 0,C 180,E1 13488.299,E2 13488.299} C_VEL
LIN {X 0,Y 334.612,Z 738.106,A -85,B 0,C 180,E1 13492.263,E2 13492.263} C_VEL
LIN {X 0,Y 334.68,Z 741.426,A -85,B 0,C 180,E1 13494.82,E2 13494.82} C_VEL
LIN {X 0,Y 334.858,Z 742.788,A -85,B 0,C 180,E1 13497.411,E2 13497.411} C_VEL
LIN {X 0,Y 335.753,Z 741.037,A -85,B 0,C 180,E1 13501.282,E2 13501.282} C_VEL
LIN {X 0,Y 337.15,Z 734.484,A -85,B 0,C 180,E1 13505.13,E2 13505.13} C_VEL
LIN {X 0,Y 339.24,Z 722.275,A -85,B 0,C 180,E1 13508.951,E2 13508.951} C_VEL
LIN {X 0,Y 341.603,Z 703.982,A -85,B 0,C 180,E1 13512.43,E2 13512.43} C_VEL
LIN {X 0,Y 343.59,Z 681.558,A -85,B 0,C 180,E1 13515.13,E2 13515.13} C_VEL
LIN {X 0,Y 344.786,Z 655.7,A -85,B 0,C 180,E1 13517.013,E2 13517.013} C_VEL
LIN {X 0,Y 345.951,Z 604.144,A -85,B 0,C 180,E1 13518.81,E2 13518.81} C_VEL
LIN {X 0,Y 345.872,Z 589.775,A -85,B 0,C 180,E1 13519.344,E2 13519.344} C_VEL
LIN {X 0,Y 337.92,Z 567.15,A -85,B 0,C 180,E1 13521.171,E2 13521.171} C_VEL
LIN {X 0,Y 329.906,Z 549.53,A -85,B 0,C 180,E1 13523.22,E2 13523.22} C_VEL
LIN {X 0,Y 329.561,Z 550.179,A -85,B 0,C 180,E1 13528.264,E2 13528.264} C_VEL
LIN {X 0,Y 332.269,Z 555.444,A -85,B 0,C 180,E1 13529.368,E2 13529.368} C_VEL
LIN {X 0,Y 343.178,Z 572.267,A -85,B 0,C 180,E1 13533.153,E2 13533.153} C_VEL
LIN {X 0,Y 357.4,Z 596.187,A -85,B 0,C 180,E1 13537.553,E2 13537.553} C_VEL
LIN {X 0,Y 372.006,Z 627.916,A -85,B 0,C 180,E1 13542.039,E2 13542.039} C_VEL
LIN {X 0,Y 375.775,Z 647.807,A -85,B 0,C 180,E1 13544.013,E2 13544.013} C_VEL
LIN {X 0,Y 367.727,Z 690.966,A -85,B 0,C 180,E1 13546.775,E2 13546.775} C_VEL
LIN {X 0,Y 359.531,Z 728.817,A -85,B 0,C 180,E1 13550.197,E2 13550.197} C_VEL
LIN {X 0,Y 351.705,Z 759.751,A -85,B 0,C 180,E1 13554.175,E2 13554.175} C_VEL
LIN {X 0,Y 344.349,Z 786.759,A -85,B 0,C 180,E1 13559.004,E2 13559.004} C_VEL
LIN {X 0,Y 338.013,Z 810.467,A -85,B 0,C 180,E1 13564.902,E2 13564.902} C_VEL
LIN {X 0,Y 333.759,Z 829.003,A -85,B 0,C 180,E1 13571.547,E2 13571.547} C_VEL
LIN {X 0,Y 332.185,Z 839.974,A -85,B 0,C 180,E1 13577.418,E2 13577.418} C_VEL
LIN {X 0,Y 331.714,Z 845.671,A -85,B 0,C 180,E1 13582.155,E2 13582.155} C_VEL
LIN {X 0,Y 331.641,Z 848.827,A -85,B 0,C 180,E1 13587.391,E2 13587.391} C_VEL
LIN {X 0,Y 331.698,Z 848.819,A -85,B 0,C 180,E1 13592.607,E2 13592.607} C_VEL
LIN {X 0,Y 331.785,Z 844.266,A -85,B 0,C 180,E1 13599.16,E2 13599.16} C_VEL
LIN {X 0,Y 332.854,Z 834.556,A -85,B 0,C 180,E1 13605.638,E2 13605.638} C_VEL
LIN {X 0,Y 332.069,Z 831.709,A -85,B 0,C 180,E1 13607.057,E2 13607.057} C_VEL
LIN {X 0,Y 327.136,Z 822.939,A -85,B 0,C 180,E1 13610.903,E2 13610.903} C_VEL
LIN {X 0,Y 327.224,Z 822.031,A -85,B 0,C 180,E1 13611.255,E2 13611.255} C_VEL
LIN {X 0,Y 332.243,Z 801.957,A -85,B 0,C 180,E1 13617.59,E2 13617.59} C_VEL
LIN {X 0,Y 338.972,Z 777.559,A -85,B 0,C 180,E1 13623.051,E2 13623.051} C_VEL
LIN {X 0,Y 346.758,Z 748.299,A -85,B 0,C 180,E1 13627.743,E2 13627.743} C_VEL
LIN {X 0,Y 354.427,Z 715.953,A -85,B 0,C 180,E1 13631.438,E2 13631.438} C_VEL
LIN {X 0,Y 363.039,Z 673.178,A -85,B 0,C 180,E1 13634.862,E2 13634.862} C_VEL
LIN {X 0,Y 367.334,Z 645.058,A -85,B 0,C 180,E1 13636.615,E2 13636.615} C_VEL
LIN {X 0,Y 361.708,Z 625.527,A -85,B 0,C 180,E1 13638.759,E2 13638.759} C_VEL
LIN {X 0,Y 347.45,Z 594.183,A -85,B 0,C 180,E1 13643.047,E2 13643.047} C_VEL
LIN {X 0,Y 339.517,Z 579.704,A -85,B 0,C 180,E1 13645.399,E2 13645.399} C_VEL
LIN {X 0,Y 338.389,Z 580.383,A -85,B 0,C 180,E1 13645.778,E2 13645.778} C_VEL
LIN {X 0,Y 344.162,Z 598.591,A -85,B 0,C 180,E1 13647.733,E2 13647.733} C_VEL
LIN {X 0,Y 342.228,Z 646.484,A -85,B 0,C 180,E1 13649.791,E2 13649.791} C_VEL
LIN {X 0,Y 340.183,Z 674.535,A -85,B 0,C 180,E1 13651.962,E2 13651.962} C_VEL
LIN {X 0,Y 337.255,Z 699.656,A -85,B 0,C 180,E1 13655.028,E2 13655.028} C_VEL
LIN {X 0,Y 334.294,Z 718.676,A -85,B 0,C 180,E1 13658.565,E2 13658.565} C_VEL
LIN {X 0,Y 331.364,Z 732.715,A -85,B 0,C 180,E1 13662.607,E2 13662.607} C_VEL
LIN {X 0,Y 329.251,Z 741.096,A -85,B 0,C 180,E1 13666.758,E2 13666.758} C_VEL
LIN {X 0,Y 328.215,Z 743.905,A -85,B 0,C 180,E1 13669.409,E2 13669.409} C_VEL
LIN {X 0,Y 327.425,Z 744.836,A -85,B 0,C 180,E1 13672.059,E2 13672.059} C_VEL
LIN {X 0,Y 326.897,Z 742.939,A -85,B 0,C 180,E1 13676.036,E2 13676.036} C_VEL
LIN {X 0,Y 326.865,Z 735.727,A -85,B 0,C 180,E1 13680.667,E2 13680.667} C_VEL
LIN {X 0,Y 327.52,Z 722.576,A -85,B 0,C 180,E1 13685.293,E2 13685.293} C_VEL
LIN {X 0,Y 328.933,Z 703.424,A -85,B 0,C 180,E1 13689.602,E2 13689.602} C_VEL
LIN {X 0,Y 330.779,Z 679.625,A -85,B 0,C 180,E1 13693.192,E2 13693.192} C_VEL
LIN {X 0,Y 332.598,Z 650.97,A -85,B 0,C 180,E1 13696.056,E2 13696.056} C_VEL
LIN {X 0,Y 333.88,Z 620.026,A -85,B 0,C 180,E1 13697.92,E2 13697.92} C_VEL
LIN {X 0,Y 333.771,Z 593.55,A -85,B 0,C 180,E1 13698.802,E2 13698.802} C_VEL
LIN {X 0,Y 322.206,Z 549.53,A -85,B 0,C 180,E1 13700.766,E2 13700.766} C_VEL
LIN {X 0,Y 321.743,Z 549.53,A -85,B 0,C 180,E1 13707.977,E2 13707.977} C_VEL
LIN {X 0,Y 321.44,Z 549.53,A -85,B 0,C 180,E1 13714.295,E2 13714.295} C_VEL
LIN {X 0,Y 321.434,Z 550.08,A -85,B 0,C 180,E1 13719.299,E2 13719.299} C_VEL
LIN {X 0,Y 324.202,Z 555.575,A -85,B 0,C 180,E1 13720.393,E2 13720.393} C_VEL
LIN {X 0,Y 338.563,Z 580.05,A -85,B 0,C 180,E1 13725.141,E2 13725.141} C_VEL
LIN {X 0,Y 352.862,Z 609.522,A -85,B 0,C 180,E1 13729.45,E2 13729.45} C_VEL
LIN {X 0,Y 360.852,Z 634.592,A -85,B 0,C 180,E1 13732.622,E2 13732.622} C_VEL
LIN {X 0,Y 354.3,Z 669.132,A -85,B 0,C 180,E1 13735.455,E2 13735.455} C_VEL
LIN {X 0,Y 346.617,Z 700.953,A -85,B 0,C 180,E1 13739.23,E2 13739.23} C_VEL
LIN {X 0,Y 339.091,Z 728.911,A -85,B 0,C 180,E1 13743.928,E2 13743.928} C_VEL
LIN {X 0,Y 332.511,Z 752.131,A -85,B 0,C 180,E1 13749.406,E2 13749.406} C_VEL
LIN {X 0,Y 327.923,Z 769.672,A -85,B 0,C 180,E1 13755.381,E2 13755.381} C_VEL
LIN {X 0,Y 325.295,Z 782.343,A -85,B 0,C 180,E1 13762,E2 13762} C_VEL
LIN {X 0,Y 324.52,Z 788.144,A -85,B 0,C 180,E1 13767.335,E2 13767.335} C_VEL
LIN {X 0,Y 324.192,Z 790.294,A -85,B 0,C 180,E1 13772.669,E2 13772.669} C_VEL
LIN {X 0,Y 324.32,Z 788.882,A -85,B 0,C 180,E1 13778.025,E2 13778.025} C_VEL
LIN {X 0,Y 325.24,Z 783.82,A -85,B 0,C 180,E1 13783.416,E2 13783.416} C_VEL
LIN {X 0,Y 328.031,Z 771.993,A -85,B 0,C 180,E1 13790.186,E2 13790.186} C_VEL
LIN {X 0,Y 332.729,Z 755.196,A -85,B 0,C 180,E1 13796.247,E2 13796.247} C_VEL
LIN {X 0,Y 339.514,Z 732.762,A -85,B 0,C 180,E1 13801.861,E2 13801.861} C_VEL
LIN {X 0,Y 347.475,Z 705.731,A -85,B 0,C 180,E1 13806.646,E2 13806.646} C_VEL
LIN {X 0,Y 355.634,Z 674.609,A -85,B 0,C 180,E1 13810.526,E2 13810.526} C_VEL
LIN {X 0,Y 362.923,Z 640.713,A -85,B 0,C 180,E1 13813.447,E2 13813.447} C_VEL
LIN {X 0,Y 363.455,Z 633.865,A -85,B 0,C 180,E1 13814.027,E2 13814.027} C_VEL
LIN {X 0,Y 354.037,Z 607.715,A -85,B 0,C 180,E1 13817.727,E2 13817.727} C_VEL
LIN {X 0,Y 339.563,Z 579.741,A -85,B 0,C 180,E1 13822.476,E2 13822.476} C_VEL
LIN {X 0,Y 327.76,Z 560.69,A -85,B 0,C 180,E1 13826.872,E2 13826.872} C_VEL
LIN {X 0,Y 324.547,Z 555.52,A -85,B 0,C 180,E1 13828.23,E2 13828.23} C_VEL
LIN {X 0,Y 321.834,Z 550.594,A -85,B 0,C 180,E1 13829.489,E2 13829.489} C_VEL
LIN {X 0,Y 321.744,Z 549.53,A -85,B 0,C 180,E1 13829.734,E2 13829.734} C_VEL
LIN {X 0,Y 321.946,Z 549.997,A -85,B 0,C 180,E1 13833.115,E2 13833.115} C_VEL
LIN {X 0,Y 332.591,Z 595.163,A -85,B 0,C 180,E1 13834.974,E2 13834.974} C_VEL
LIN {X 0,Y 331.85,Z 643.761,A -85,B 0,C 180,E1 13836.458,E2 13836.458} C_VEL
LIN {X 0,Y 330.947,Z 670.591,A -85,B 0,C 180,E1 13838.248,E2 13838.248} C_VEL
LIN {X 0,Y 329.65,Z 693.951,A -85,B 0,C 180,E1 13840.81,E2 13840.81} C_VEL
LIN {X 0,Y 328.091,Z 714.97,A -85,B 0,C 180,E1 13844.342,E2 13844.342} C_VEL
LIN {X 0,Y 327.17,Z 730.278,A -85,B 0,C 180,E1 13848.352,E2 13848.352} C_VEL
LIN {X 0,Y 326.802,Z 739.292,A -85,B 0,C 180,E1 13852.253,E2 13852.253} C_VEL
LIN {X 0,Y 326.898,Z 742.562,A -85,B 0,C 180,E1 13854.697,E2 13854.697} C_VEL
LIN {X 0,Y 327.071,Z 744.158,A -85,B 0,C 180,E1 13857.35,E2 13857.35} C_VEL
LIN {X 0,Y 328.012,Z 742.693,A -85,B 0,C 180,E1 13861.312,E2 13861.312} C_VEL
LIN {X 0,Y 329.519,Z 736.516,A -85,B 0,C 180,E1 13865.249,E2 13865.249} C_VEL
LIN {X 0,Y 331.757,Z 724.623,A -85,B 0,C 180,E1 13869.154,E2 13869.154} C_VEL
LIN {X 0,Y 334.264,Z 706.933,A -85,B 0,C 180,E1 13872.708,E2 13872.708} C_VEL
LIN {X 0,Y 336.507,Z 684.009,A -85,B 0,C 180,E1 13875.602,E2 13875.602} C_VEL
LIN {X 0,Y 337.876,Z 658.615,A -85,B 0,C 180,E1 13877.54,E2 13877.54} C_VEL
LIN {X 0,Y 338.954,Z 612.103,A -85,B 0,C 180,E1 13879.294,E2 13879.294} C_VEL
LIN {X 0,Y 339.169,Z 591.398,A -85,B 0,C 180,E1 13880.046,E2 13880.046} C_VEL
LIN {X 0,Y 331.184,Z 568.816,A -85,B 0,C 180,E1 13882.041,E2 13882.041} C_VEL
LIN {X 0,Y 321.845,Z 549.53,A -85,B 0,C 180,E1 13884.564,E2 13884.564} C_VEL
LIN {X 0,Y 321.758,Z 550.328,A -85,B 0,C 180,E1 13885.836,E2 13885.836} C_VEL
LIN {X 0,Y 324.494,Z 555.535,A -85,B 0,C 180,E1 13887.078,E2 13887.078} C_VEL
LIN {X 0,Y 326.849,Z 559.088,A -85,B 0,C 180,E1 13888.038,E2 13888.038} C_VEL
LIN {X 0,Y 338.313,Z 576.434,A -85,B 0,C 180,E1 13892.262,E2 13892.262} C_VEL
LIN {X 0,Y 353.246,Z 602.838,A -85,B 0,C 180,E1 13897.203,E2 13897.203} C_VEL
LIN {X 0,Y 366.606,Z 632.875,A -85,B 0,C 180,E1 13901.578,E2 13901.578} C_VEL
LIN {X 0,Y 369.48,Z 650.08,A -85,B 0,C 180,E1 13903.312,E2 13903.312} C_VEL
LIN {X 0,Y 361.411,Z 691.486,A -85,B 0,C 180,E1 13906.034,E2 13906.034} C_VEL
LIN {X 0,Y 353.21,Z 728.082,A -85,B 0,C 180,E1 13909.381,E2 13909.381} C_VEL
LIN {X 0,Y 344.834,Z 759.518,A -85,B 0,C 180,E1 13913.481,E2 13913.481} C_VEL
LIN {X 0,Y 336.775,Z 787.746,A -85,B 0,C 180,E1 13918.669,E2 13918.669} C_VEL
LIN {X 0,Y 330.291,Z 810.778,A -85,B 0,C 180,E1 13924.636,E2 13924.636} C_VEL
LIN {X 0,Y 326.039,Z 828.276,A -85,B 0,C 180,E1 13931.093,E2 13931.093} C_VEL
LIN {X 0,Y 324.251,Z 840.163,A -85,B 0,C 180,E1 13937.744,E2 13937.744} C_VEL
LIN {X 0,Y 323.834,Z 844.972,A -85,B 0,C 180,E1 13941.963,E2 13941.963} C_VEL
LIN {X 0,Y 323.757,Z 848.122,A -85,B 0,C 180,E1 13947.328,E2 13947.328} C_VEL
LIN {X 0,Y 323.813,Z 848.103,A -85,B 0,C 180,E1 13952.671,E2 13952.671} C_VEL
LIN {X 0,Y 323.904,Z 843.515,A -85,B 0,C 180,E1 13959.385,E2 13959.385} C_VEL
LIN {X 0,Y 325.119,Z 833.465,A -85,B 0,C 180,E1 13966.171,E2 13966.171} C_VEL
LIN {X 0,Y 327.224,Z 822.031,A -85,B 0,C 180,E1 13971.255,E2 13971.255} C_VEL
LIN {X 0,Y 325.103,Z 814.645,A -85,B 0,C 180,E1 13974.026,E2 13974.026} C_VEL
LIN {X 0,Y 323.396,Z 806.365,A -85,B 0,C 180,E1 13976.752,E2 13976.752} C_VEL
LIN {X 0,Y 330.522,Z 781.902,A -85,B 0,C 180,E1 13982.736,E2 13982.736} C_VEL
LIN {X 0,Y 338.594,Z 753.148,A -85,B 0,C 180,E1 13987.716,E2 13987.716} C_VEL
LIN {X 0,Y 346.719,Z 721.357,A -85,B 0,C 180,E1 13991.628,E2 13991.628} C_VEL
LIN {X 0,Y 355.367,Z 680.544,A -85,B 0,C 180,E1 13995.128,E2 13995.128} C_VEL
LIN {X 0,Y 361.042,Z 647.928,A -85,B 0,C 180,E1 13997.227,E2 13997.227} C_VEL
LIN {X 0,Y 355.655,Z 628.871,A -85,B 0,C 180,E1 13999.428,E2 13999.428} C_VEL
LIN {X 0,Y 342.07,Z 598.518,A -85,B 0,C 180,E1 14003.756,E2 14003.756} C_VEL
LIN {X 0,Y 337.152,Z 589.247,A -85,B 0,C 180,E1 14005.294,E2 14005.294} C_VEL
LIN {X 0,Y 335.44,Z 590.155,A -85,B 0,C 180,E1 14005.764,E2 14005.764} C_VEL
LIN {X 0,Y 338.318,Z 602.498,A -85,B 0,C 180,E1 14006.973,E2 14006.973} C_VEL
LIN {X 0,Y 335.921,Z 649.282,A -85,B 0,C 180,E1 14009.093,E2 14009.093} C_VEL
LIN {X 0,Y 333.6,Z 677.233,A -85,B 0,C 180,E1 14011.358,E2 14011.358} C_VEL
LIN {X 0,Y 330.578,Z 700.804,A -85,B 0,C 180,E1 14014.307,E2 14014.307} C_VEL
LIN {X 0,Y 327.333,Z 719.872,A -85,B 0,C 180,E1 14017.893,E2 14017.893} C_VEL
LIN {X 0,Y 324.205,Z 733.857,A -85,B 0,C 180,E1 14021.943,E2 14021.943} C_VEL
LIN {X 0,Y 321.714,Z 742.792,A -85,B 0,C 180,E1 14026.442,E2 14026.442} C_VEL
LIN {X 0,Y 320.586,Z 745.509,A -85,B 0,C 180,E1 14029.154,E2 14029.154} C_VEL
LIN {X 0,Y 319.576,Z 746.294,A -85,B 0,C 180,E1 14032.614,E2 14032.614} C_VEL
LIN {X 0,Y 319.027,Z 742.76,A -85,B 0,C 180,E1 14037.295,E2 14037.295} C_VEL
LIN {X 0,Y 319.177,Z 733.783,A -85,B 0,C 180,E1 14042.038,E2 14042.038} C_VEL
LIN {X 0,Y 320.082,Z 718.429,A -85,B 0,C 180,E1 14046.775,E2 14046.775} C_VEL
LIN {X 0,Y 321.673,Z 698.459,A -85,B 0,C 180,E1 14050.822,E2 14050.822} C_VEL
LIN {X 0,Y 323.521,Z 674.288,A -85,B 0,C 180,E1 14054.181,E2 14054.181} C_VEL
LIN {X 0,Y 325.291,Z 645.273,A -85,B 0,C 180,E1 14056.841,E2 14056.841} C_VEL
LIN {X 0,Y 326.39,Z 612.43,A -85,B 0,C 180,E1 14058.579,E2 14058.579} C_VEL
LIN {X 0,Y 325.795,Z 593.499,A -85,B 0,C 180,E1 14059.198,E2 14059.198} C_VEL
LIN {X 0,Y 314.217,Z 549.53,A -85,B 0,C 180,E1 14061.332,E2 14061.332} C_VEL
LIN {X 0,Y 313.697,Z 549.53,A -85,B 0,C 180,E1 14068.761,E2 14068.761} C_VEL
LIN {X 0,Y 313.476,Z 549.532,A -85,B 0,C 180,E1 14077.079,E2 14077.079} C_VEL
LIN {X 0,Y 315.76,Z 555.064,A -85,B 0,C 180,E1 14078.15,E2 14078.15} C_VEL
LIN {X 0,Y 321.996,Z 564.937,A -85,B 0,C 180,E1 14080.51,E2 14080.51} C_VEL
LIN {X 0,Y 334.945,Z 587.452,A -85,B 0,C 180,E1 14084.897,E2 14084.897} C_VEL
LIN {X 0,Y 347.857,Z 615.29,A -85,B 0,C 180,E1 14089.047,E2 14089.047} C_VEL
LIN {X 0,Y 354.541,Z 637.333,A -85,B 0,C 180,E1 14091.96,E2 14091.96} C_VEL
LIN {X 0,Y 347.595,Z 671.883,A -85,B 0,C 180,E1 14094.881,E2 14094.881} C_VEL
LIN {X 0,Y 339.644,Z 703.11,A -85,B 0,C 180,E1 14098.714,E2 14098.714} C_VEL
LIN {X 0,Y 332.028,Z 729.891,A -85,B 0,C 180,E1 14103.33,E2 14103.33} C_VEL
LIN {X 0,Y 325.142,Z 753.027,A -85,B 0,C 180,E1 14108.917,E2 14108.917} C_VEL
LIN {X 0,Y 320.299,Z 770.541,A -85,B 0,C 180,E1 14115.04,E2 14115.04} C_VEL
LIN {X 0,Y 317.503,Z 783.119,A -85,B 0,C 180,E1 14121.802,E2 14121.802} C_VEL
LIN {X 0,Y 316.662,Z 788.888,A -85,B 0,C 180,E1 14127.269,E2 14127.269} C_VEL
LIN {X 0,Y 316.345,Z 791.005,A -85,B 0,C 180,E1 14132.735,E2 14132.735} C_VEL
LIN {X 0,Y 316.653,Z 788.657,A -85,B 0,C 180,E1 14139.603,E2 14139.603} C_VEL
LIN {X 0,Y 318.074,Z 781.584,A -85,B 0,C 180,E1 14145.833,E2 14145.833} C_VEL
LIN {X 0,Y 321.337,Z 769.418,A -85,B 0,C 180,E1 14152.07,E2 14152.07} C_VEL
LIN {X 0,Y 326.986,Z 751.077,A -85,B 0,C 180,E1 14158.262,E2 14158.262} C_VEL
LIN {X 0,Y 334.768,Z 727.114,A -85,B 0,C 180,E1 14163.852,E2 14163.852} C_VEL
LIN {X 0,Y 343.425,Z 698.557,A -85,B 0,C 180,E1 14168.544,E2 14168.544} C_VEL
LIN {X 0,Y 351.504,Z 667.482,A -85,B 0,C 180,E1 14172.134,E2 14172.134} C_VEL
LIN {X 0,Y 357.418,Z 636.96,A -85,B 0,C 180,E1 14174.705,E2 14174.705} C_VEL
LIN {X 0,Y 348.046,Z 610.475,A -85,B 0,C 180,E1 14178.643,E2 14178.643} C_VEL
LIN {X 0,Y 334.409,Z 584.064,A -85,B 0,C 180,E1 14183.373,E2 14183.373} C_VEL
LIN {X 0,Y 321.632,Z 562.646,A -85,B 0,C 180,E1 14188.522,E2 14188.522} C_VEL
LIN {X 0,Y 316.787,Z 555.643,A -85,B 0,C 180,E1 14190.734,E2 14190.734} C_VEL
LIN {X 0,Y 314.035,Z 550.709,A -85,B 0,C 180,E1 14192.187,E2 14192.187} C_VEL
LIN {X 0,Y 313.975,Z 549.53,A -85,B 0,C 180,E1 14192.634,E2 14192.634} C_VEL
LIN {X 0,Y 325.018,Z 593.952,A -85,B 0,C 180,E1 14194.585,E2 14194.585} C_VEL
LIN {X 0,Y 324.121,Z 645.946,A -85,B 0,C 180,E1 14196.227,E2 14196.227} C_VEL
LIN {X 0,Y 323.147,Z 673.459,A -85,B 0,C 180,E1 14198.159,E2 14198.159} C_VEL
LIN {X 0,Y 321.699,Z 697.858,A -85,B 0,C 180,E1 14201.002,E2 14201.002} C_VEL
LIN {X 0,Y 320.202,Z 717.689,A -85,B 0,C 180,E1 14204.549,E2 14204.549} C_VEL
LIN {X 0,Y 319.338,Z 731.786,A -85,B 0,C 180,E1 14208.408,E2 14208.408} C_VEL
LIN {X 0,Y 319.002,Z 741.612,A -85,B 0,C 180,E1 14212.92,E2 14212.92} C_VEL
LIN {X 0,Y 319.298,Z 745.514,A -85,B 0,C 180,E1 14217.285,E2 14217.285} C_VEL
LIN {X 0,Y 320.295,Z 744.381,A -85,B 0,C 180,E1 14221.344,E2 14221.344} C_VEL
LIN {X 0,Y 321.908,Z 738.495,A -85,B 0,C 180,E1 14225.374,E2 14225.374} C_VEL
LIN {X 0,Y 324.301,Z 727.065,A -85,B 0,C 180,E1 14229.367,E2 14229.367} C_VEL
LIN {X 0,Y 326.98,Z 709.913,A -85,B 0,C 180,E1 14232.996,E2 14232.996} C_VEL
LIN {X 0,Y 329.228,Z 689.623,A -85,B 0,C 180,E1 14235.766,E2 14235.766} C_VEL
LIN {X 0,Y 330.976,Z 663.189,A -85,B 0,C 180,E1 14238.004,E2 14238.004} C_VEL
LIN {X 0,Y 331.805,Z 627.834,A -85,B 0,C 180,E1 14239.521,E2 14239.521} C_VEL
LIN {X 0,Y 332.88,Z 593.853,A -85,B 0,C 180,E1 14240.739,E2 14240.739} C_VEL
LIN {X 0,Y 325.382,Z 572.661,A -85,B 0,C 180,E1 14242.75,E2 14242.75} C_VEL
LIN {X 0,Y 317.731,Z 557.144,A -85,B 0,C 180,E1 14244.982,E2 14244.982} C_VEL
LIN {X 0,Y 324.289,Z 566.961,A -85,B 0,C 180,E1 14247.843,E2 14247.843} C_VEL
LIN {X 0,Y 337.671,Z 587.97,A -85,B 0,C 180,E1 14252.898,E2 14252.898} C_VEL
LIN {X 0,Y 352.449,Z 616.309,A -85,B 0,C 180,E1 14257.998,E2 14257.998} C_VEL
LIN {X 0,Y 361.425,Z 639.353,A -85,B 0,C 180,E1 14261.269,E2 14261.269} C_VEL
LIN {X 0,Y 363.295,Z 651.863,A -85,B 0,C 180,E1 14262.569,E2 14262.569} C_VEL
LIN {X 0,Y 354.753,Z 693.923,A -85,B 0,C 180,E1 14265.417,E2 14265.417} C_VEL
LIN {X 0,Y 346.212,Z 729.997,A -85,B 0,C 180,E1 14268.829,E2 14268.829} C_VEL
LIN {X 0,Y 337.524,Z 761.036,A -85,B 0,C 180,E1 14273.035,E2 14273.035} C_VEL
LIN {X 0,Y 329.234,Z 788.578,A -85,B 0,C 180,E1 14278.304,E2 14278.304} C_VEL
LIN {X 0,Y 322.558,Z 811.1,A -85,B 0,C 180,E1 14284.355,E2 14284.355} C_VEL
LIN {X 0,Y 318.346,Z 827.548,A -85,B 0,C 180,E1 14290.618,E2 14290.618} C_VEL
LIN {X 0,Y 316.38,Z 839.446,A -85,B 0,C 180,E1 14297.435,E2 14297.435} C_VEL
LIN {X 0,Y 315.953,Z 844.271,A -85,B 0,C 180,E1 14301.761,E2 14301.761} C_VEL
LIN {X 0,Y 315.888,Z 847.419,A -85,B 0,C 180,E1 14307.261,E2 14307.261} C_VEL
LIN {X 0,Y 315.932,Z 847.387,A -85,B 0,C 180,E1 14312.738,E2 14312.738} C_VEL
LIN {X 0,Y 316.041,Z 842.761,A -85,B 0,C 180,E1 14319.621,E2 14319.621} C_VEL
LIN {X 0,Y 317.335,Z 832.647,A -85,B 0,C 180,E1 14326.579,E2 14326.579} C_VEL
LIN {X 0,Y 320.73,Z 816.658,A -85,B 0,C 180,E1 14333.458,E2 14333.458} C_VEL
LIN {X 0,Y 323.396,Z 806.365,A -85,B 0,C 180,E1 14336.752,E2 14336.752} C_VEL
LIN {X 0,Y 322.096,Z 797.441,A -85,B 0,C 180,E1 14339.423,E2 14339.423} C_VEL
LIN {X 0,Y 321.364,Z 787.689,A -85,B 0,C 180,E1 14342.025,E2 14342.025} C_VEL
LIN {X 0,Y 329.662,Z 759.976,A -85,B 0,C 180,E1 14347.342,E2 14347.342} C_VEL
LIN {X 0,Y 338.44,Z 728.257,A -85,B 0,C 180,E1 14351.631,E2 14351.631} C_VEL
LIN {X 0,Y 346.788,Z 691.737,A -85,B 0,C 180,E1 14355.087,E2 14355.087} C_VEL
LIN {X 0,Y 354.65,Z 649.874,A -85,B 0,C 180,E1 14357.964,E2 14357.964} C_VEL
LIN {X 0,Y 349.403,Z 631.683,A -85,B 0,C 180,E1 14360.174,E2 14360.174} C_VEL
LIN {X 0,Y 335.98,Z 601.316,A -85,B 0,C 180,E1 14364.721,E2 14364.721} C_VEL
LIN {X 0,Y 334.096,Z 598.969,A -85,B 0,C 180,E1 14365.258,E2 14365.258} C_VEL
LIN {X 0,Y 332.174,Z 600.586,A -85,B 0,C 180,E1 14365.726,E2 14365.726} C_VEL
LIN {X 0,Y 332.496,Z 607.638,A -85,B 0,C 180,E1 14366.197,E2 14366.197} C_VEL
LIN {X 0,Y 329.849,Z 651.643,A -85,B 0,C 180,E1 14368.312,E2 14368.312} C_VEL
LIN {X 0,Y 327.132,Z 680.268,A -85,B 0,C 180,E1 14370.729,E2 14370.729} C_VEL
LIN {X 0,Y 323.483,Z 705.413,A -85,B 0,C 180,E1 14374.073,E2 14374.073} C_VEL
LIN {X 0,Y 319.922,Z 723.844,A -85,B 0,C 180,E1 14377.837,E2 14377.837} C_VEL
LIN {X 0,Y 316.617,Z 736.86,A -85,B 0,C 180,E1 14381.941,E2 14381.941} C_VEL
LIN {X 0,Y 314.202,Z 744.523,A -85,B 0,C 180,E1 14386.112,E2 14386.112} C_VEL
LIN {X 0,Y 312.963,Z 747.14,A -85,B 0,C 180,E1 14388.886,E2 14388.886} C_VEL
LIN {X 0,Y 312.025,Z 747.902,A -85,B 0,C 180,E1 14391.664,E2 14391.664} C_VEL
LIN {X 0,Y 311.34,Z 745.698,A -85,B 0,C 180,E1 14395.837,E2 14395.837} C_VEL
LIN {X 0,Y 311.227,Z 738.115,A -85,B 0,C 180,E1 14400.701,E2 14400.701} C_VEL
LIN {X 0,Y 311.928,Z 724.445,A -85,B 0,C 180,E1 14405.559,E2 14405.559} C_VEL
LIN {X 0,Y 313.383,Z 705.546,A -85,B 0,C 180,E1 14409.918,E2 14409.918} C_VEL
LIN {X 0,Y 315.315,Z 681.473,A -85,B 0,C 180,E1 14413.675,E2 14413.675} C_VEL
LIN {X 0,Y 317.214,Z 653.33,A -85,B 0,C 180,E1 14416.591,E2 14416.591} C_VEL
LIN {X 0,Y 318.615,Z 621.143,A -85,B 0,C 180,E1 14418.601,E2 14418.601} C_VEL
LIN {X 0,Y 318.405,Z 595.724,A -85,B 0,C 180,E1 14419.498,E2 14419.498} C_VEL
LIN {X 0,Y 306.246,Z 549.53,A -85,B 0,C 180,E1 14421.789,E2 14421.789} C_VEL
LIN {X 0,Y 305.742,Z 549.53,A -85,B 0,C 180,E1 14429.582,E2 14429.582} C_VEL
LIN {X 0,Y 305.581,Z 550.049,A -85,B 0,C 180,E1 14434.68,E2 14434.68} C_VEL
LIN {X 0,Y 308.242,Z 555.452,A -85,B 0,C 180,E1 14435.986,E2 14435.986} C_VEL
LIN {X 0,Y 317.432,Z 569.894,A -85,B 0,C 180,E1 14439.728,E2 14439.728} C_VEL
LIN {X 0,Y 331.386,Z 594.876,A -85,B 0,C 180,E1 14444.675,E2 14444.675} C_VEL
LIN {X 0,Y 342.893,Z 621.244,A -85,B 0,C 180,E1 14448.686,E2 14448.686} C_VEL
LIN {X 0,Y 348.177,Z 640.263,A -85,B 0,C 180,E1 14451.282,E2 14451.282} C_VEL
LIN {X 0,Y 340.899,Z 674.513,A -85,B 0,C 180,E1 14454.281,E2 14454.281} C_VEL
LIN {X 0,Y 332.67,Z 705.275,A -85,B 0,C 180,E1 14458.172,E2 14458.172} C_VEL
LIN {X 0,Y 324.536,Z 732.419,A -85,B 0,C 180,E1 14463.038,E2 14463.038} C_VEL
LIN {X 0,Y 317.471,Z 755.046,A -85,B 0,C 180,E1 14468.748,E2 14468.748} C_VEL
LIN {X 0,Y 312.475,Z 772.157,A -85,B 0,C 180,E1 14475.009,E2 14475.009} C_VEL
LIN {X 0,Y 309.718,Z 783.896,A -85,B 0,C 180,E1 14481.595,E2 14481.595} C_VEL
LIN {X 0,Y 308.819,Z 789.63,A -85,B 0,C 180,E1 14487.199,E2 14487.199} C_VEL
LIN {X 0,Y 308.487,Z 791.717,A -85,B 0,C 180,E1 14492.805,E2 14492.805} C_VEL
LIN {X 0,Y 308.848,Z 789.331,A -85,B 0,C 180,E1 14499.848,E2 14499.848} C_VEL
LIN {X 0,Y 310.651,Z 781.181,A -85,B 0,C 180,E1 14506.948,E2 14506.948} C_VEL
LIN {X 0,Y 314.55,Z 767.61,A -85,B 0,C 180,E1 14513.622,E2 14513.622} C_VEL
LIN {X 0,Y 320.76,Z 749.179,A -85,B 0,C 180,E1 14519.662,E2 14519.662} C_VEL
LIN {X 0,Y 328.768,Z 725.724,A -85,B 0,C 180,E1 14525.015,E2 14525.015} C_VEL
LIN {X 0,Y 337.8,Z 696.936,A -85,B 0,C 180,E1 14529.682,E2 14529.682} C_VEL
LIN {X 0,Y 346.46,Z 664.815,A -85,B 0,C 180,E1 14533.32,E2 14533.32} C_VEL
LIN {X 0,Y 351.435,Z 640.364,A -85,B 0,C 180,E1 14535.366,E2 14535.366} C_VEL
LIN {X 0,Y 342.866,Z 615.105,A -85,B 0,C 180,E1 14539.283,E2 14539.283} C_VEL
LIN {X 0,Y 329.649,Z 588.74,A -85,B 0,C 180,E1 14544.184,E2 14544.184} C_VEL
LIN {X 0,Y 317.906,Z 569.019,A -85,B 0,C 180,E1 14549.141,E2 14549.141} C_VEL
LIN {X 0,Y 313.557,Z 562.482,A -85,B 0,C 180,E1 14551.225,E2 14551.225} C_VEL
LIN {X 0,Y 309.579,Z 563.152,A -85,B 0,C 180,E1 14552.834,E2 14552.834} C_VEL
LIN {X 0,Y 317.336,Z 596.76,A -85,B 0,C 180,E1 14554.286,E2 14554.286} C_VEL
LIN {X 0,Y 316.451,Z 647.537,A -85,B 0,C 180,E1 14555.955,E2 14555.955} C_VEL
LIN {X 0,Y 315.388,Z 675.69,A -85,B 0,C 180,E1 14558.015,E2 14558.015} C_VEL
LIN {X 0,Y 313.796,Z 700.53,A -85,B 0,C 180,E1 14561.052,E2 14561.052} C_VEL
LIN {X 0,Y 312.325,Z 720.742,A -85,B 0,C 180,E1 14564.884,E2 14564.884} C_VEL
LIN {X 0,Y 311.444,Z 734.264,A -85,B 0,C 180,E1 14568.818,E2 14568.818} C_VEL
LIN {X 0,Y 311.229,Z 743.35,A -85,B 0,C 180,E1 14573.274,E2 14573.274} C_VEL
LIN {X 0,Y 311.506,Z 746.853,A -85,B 0,C 180,E1 14577.217,E2 14577.217} C_VEL
LIN {X 0,Y 312.581,Z 746.062,A -85,B 0,C 180,E1 14581.377,E2 14581.377} C_VEL
LIN {X 0,Y 314.293,Z 740.543,A -85,B 0,C 180,E1 14585.504,E2 14585.504} C_VEL
LIN {X 0,Y 316.839,Z 729.54,A -85,B 0,C 180,E1 14589.589,E2 14589.589} C_VEL
LIN {X 0,Y 319.707,Z 713.007,A -85,B 0,C 180,E1 14593.297,E2 14593.297} C_VEL
LIN {X 0,Y 322.302,Z 691.971,A -85,B 0,C 180,E1 14596.309,E2 14596.309} C_VEL
LIN {X 0,Y 324.191,Z 666.464,A -85,B 0,C 180,E1 14598.569,E2 14598.569} C_VEL
LIN {X 0,Y 325.136,Z 634.405,A -85,B 0,C 180,E1 14600.082,E2 14600.082} C_VEL
LIN {X 0,Y 326.515,Z 595.701,A -85,B 0,C 180,E1 14601.534,E2 14601.534} C_VEL
LIN {X 0,Y 319.121,Z 574.993,A -85,B 0,C 180,E1 14603.674,E2 14603.674} C_VEL
LIN {X 0,Y 315.312,Z 566.599,A -85,B 0,C 180,E1 14604.924,E2 14604.924} C_VEL
LIN {X 0,Y 317.27,Z 567.99,A -85,B 0,C 180,E1 14605.709,E2 14605.709} C_VEL
LIN {X 0,Y 327.918,Z 584.591,A -85,B 0,C 180,E1 14610.213,E2 14610.213} C_VEL
LIN {X 0,Y 341.916,Z 609.766,A -85,B 0,C 180,E1 14615.454,E2 14615.454} C_VEL
LIN {X 0,Y 354.725,Z 639.674,A -85,B 0,C 180,E1 14620.216,E2 14620.216} C_VEL
LIN {X 0,Y 356.978,Z 654.966,A -85,B 0,C 180,E1 14621.877,E2 14621.877} C_VEL
LIN {X 0,Y 347.704,Z 698.223,A -85,B 0,C 180,E1 14624.925,E2 14624.925} C_VEL
LIN {X 0,Y 339.467,Z 731.197,A -85,B 0,C 180,E1 14628.174,E2 14628.174} C_VEL
LIN {X 0,Y 330.621,Z 761.315,A -85,B 0,C 180,E1 14632.372,E2 14632.372} C_VEL
LIN {X 0,Y 321.964,Z 788.596,A -85,B 0,C 180,E1 14637.73,E2 14637.73} C_VEL
LIN {X 0,Y 314.848,Z 811.406,A -85,B 0,C 180,E1 14644.062,E2 14644.062} C_VEL
LIN {X 0,Y 310.154,Z 829.015,A -85,B 0,C 180,E1 14651.203,E2 14651.203} C_VEL
LIN {X 0,Y 308.385,Z 840.023,A -85,B 0,C 180,E1 14658.113,E2 14658.113} C_VEL
LIN {X 0,Y 307.938,Z 845.537,A -85,B 0,C 180,E1 14664.374,E2 14664.374} C_VEL
LIN {X 0,Y 308.306,Z 847.131,A -85,B 0,C 180,E1 14669.999,E2 14669.999} C_VEL
LIN {X 0,Y 308.016,Z 844.481,A -85,B 0,C 180,E1 14677.035,E2 14677.035} C_VEL
LIN {X 0,Y 308.821,Z 836.588,A -85,B 0,C 180,E1 14684.143,E2 14684.143} C_VEL
LIN {X 0,Y 311.033,Z 824.464,A -85,B 0,C 180,E1 14690.596,E2 14690.596} C_VEL
LIN {X 0,Y 315.974,Z 805.581,A -85,B 0,C 180,E1 14697.368,E2 14697.368} C_VEL
LIN {X 0,Y 321.364,Z 787.689,A -85,B 0,C 180,E1 14702.025,E2 14702.025} C_VEL
LIN {X 0,Y 321.048,Z 777.372,A -85,B 0,C 180,E1 14704.553,E2 14704.553} C_VEL
LIN {X 0,Y 320.852,Z 766.162,A -85,B 0,C 180,E1 14706.966,E2 14706.966} C_VEL
LIN {X 0,Y 329.537,Z 736.586,A -85,B 0,C 180,E1 14711.406,E2 14711.406} C_VEL
LIN {X 0,Y 338.153,Z 702.483,A -85,B 0,C 180,E1 14714.995,E2 14714.995} C_VEL
LIN {X 0,Y 347.69,Z 657.508,A -85,B 0,C 180,E1 14718.311,E2 14718.311} C_VEL
LIN {X 0,Y 347.976,Z 650.15,A -85,B 0,C 180,E1 14718.911,E2 14718.911} C_VEL
LIN {X 0,Y 339.435,Z 624.817,A -85,B 0,C 180,E1 14722.354,E2 14722.354} C_VEL
LIN {X 0,Y 332.107,Z 609.595,A -85,B 0,C 180,E1 14724.881,E2 14724.881} C_VEL
LIN {X 0,Y 326.518,Z 616.49,A -85,B 0,C 180,E1 14725.525,E2 14725.525} C_VEL
LIN {X 0,Y 323.854,Z 655.361,A -85,B 0,C 180,E1 14727.562,E2 14727.562} C_VEL
LIN {X 0,Y 320.632,Z 684.228,A -85,B 0,C 180,E1 14730.154,E2 14730.154} C_VEL
LIN {X 0,Y 316.788,Z 707.996,A -85,B 0,C 180,E1 14733.482,E2 14733.482} C_VEL
LIN {X 0,Y 312.903,Z 726.031,A -85,B 0,C 180,E1 14737.313,E2 14737.313} C_VEL
LIN {X 0,Y 309.321,Z 738.861,A -85,B 0,C 180,E1 14741.519,E2 14741.519} C_VEL
LIN {X 0,Y 306.707,Z 746.302,A -85,B 0,C 180,E1 14745.765,E2 14745.765} C_VEL
LIN {X 0,Y 305.368,Z 748.779,A -85,B 0,C 180,E1 14748.606,E2 14748.606} C_VEL
LIN {X 0,Y 303.877,Z 748.887,A -85,B 0,C 180,E1 14753.35,E2 14753.35} C_VEL
LIN {X 0,Y 303.384,Z 743.314,A -85,B 0,C 180,E1 14758.581,E2 14758.581} C_VEL
LIN {X 0,Y 303.749,Z 732.119,A -85,B 0,C 180,E1 14763.567,E2 14763.567} C_VEL
LIN {X 0,Y 304.892,Z 715.452,A -85,B 0,C 180,E1 14768.222,E2 14768.222} C_VEL
LIN {X 0,Y 306.7,Z 692.841,A -85,B 0,C 180,E1 14772.437,E2 14772.437} C_VEL
LIN {X 0,Y 308.799,Z 666.13,A -85,B 0,C 180,E1 14775.78,E2 14775.78} C_VEL
LIN {X 0,Y 310.39,Z 636.387,A -85,B 0,C 180,E1 14778.175,E2 14778.175} C_VEL
LIN {X 0,Y 311.427,Z 601.955,A -85,B 0,C 180,E1 14779.66,E2 14779.66} C_VEL
LIN {X 0,Y 298.286,Z 549.53,A -85,B 0,C 180,E1 14782.228,E2 14782.228} C_VEL
LIN {X 0,Y 297.712,Z 549.53,A -85,B 0,C 180,E1 14790.485,E2 14790.485} C_VEL
LIN {X 0,Y 297.621,Z 549.951,A -85,B 0,C 180,E1 14791.846,E2 14791.846} C_VEL
LIN {X 0,Y 300.263,Z 555.4,A -85,B 0,C 180,E1 14793.352,E2 14793.352} C_VEL
LIN {X 0,Y 302.447,Z 558.291,A -85,B 0,C 180,E1 14794.37,E2 14794.37} C_VEL
LIN {X 0,Y 314.113,Z 577.334,A -85,B 0,C 180,E1 14799.445,E2 14799.445} C_VEL
LIN {X 0,Y 327.176,Z 601.333,A -85,B 0,C 180,E1 14804.26,E2 14804.26} C_VEL
LIN {X 0,Y 337.995,Z 627.729,A -85,B 0,C 180,E1 14808.397,E2 14808.397} C_VEL
LIN {X 0,Y 341.76,Z 643.954,A -85,B 0,C 180,E1 14810.639,E2 14810.639} C_VEL
LIN {X 0,Y 333.864,Z 678.501,A -85,B 0,C 180,E1 14813.81,E2 14813.81} C_VEL
LIN {X 0,Y 325.408,Z 708.479,A -85,B 0,C 180,E1 14817.769,E2 14817.769} C_VEL
LIN {X 0,Y 317.052,Z 734.939,A -85,B 0,C 180,E1 14822.733,E2 14822.733} C_VEL
LIN {X 0,Y 309.758,Z 757.025,A -85,B 0,C 180,E1 14828.568,E2 14828.568} C_VEL
LIN {X 0,Y 304.584,Z 774.113,A -85,B 0,C 180,E1 14835.134,E2 14835.134} C_VEL
LIN {X 0,Y 301.933,Z 784.673,A -85,B 0,C 180,E1 14841.376,E2 14841.376} C_VEL
LIN {X 0,Y 300.962,Z 790.372,A -85,B 0,C 180,E1 14847.126,E2 14847.126} C_VEL
LIN {X 0,Y 300.613,Z 792.43,A -85,B 0,C 180,E1 14852.878,E2 14852.878} C_VEL
LIN {X 0,Y 301.04,Z 790.006,A -85,B 0,C 180,E1 14860.106,E2 14860.106} C_VEL
LIN {X 0,Y 303.009,Z 781.841,A -85,B 0,C 180,E1 14867.388,E2 14867.388} C_VEL
LIN {X 0,Y 307.084,Z 768.614,A -85,B 0,C 180,E1 14874.07,E2 14874.07} C_VEL
LIN {X 0,Y 313.732,Z 749.977,A -85,B 0,C 180,E1 14880.334,E2 14880.334} C_VEL
LIN {X 0,Y 322.232,Z 726.298,A -85,B 0,C 180,E1 14885.835,E2 14885.835} C_VEL
LIN {X 0,Y 331.191,Z 699.179,A -85,B 0,C 180,E1 14890.327,E2 14890.327} C_VEL
LIN {X 0,Y 340.317,Z 666.915,A -85,B 0,C 180,E1 14894.082,E2 14894.082} C_VEL
LIN {X 0,Y 345.372,Z 643.252,A -85,B 0,C 180,E1 14896.126,E2 14896.126} C_VEL
LIN {X 0,Y 336.801,Z 617.663,A -85,B 0,C 180,E1 14900.314,E2 14900.314} C_VEL
LIN {X 0,Y 324.335,Z 592.505,A -85,B 0,C 180,E1 14905.246,E2 14905.246} C_VEL
LIN {X 0,Y 313.958,Z 574.969,A -85,B 0,C 180,E1 14909.881,E2 14909.881} C_VEL
LIN {X 0,Y 310.713,Z 570.172,A -85,B 0,C 180,E1 14911.487,E2 14911.487} C_VEL
LIN {X 0,Y 306.117,Z 576.351,A -85,B 0,C 180,E1 14912.559,E2 14912.559} C_VEL
LIN {X 0,Y 305.232,Z 576.955,A -85,B 0,C 180,E1 14913.041,E2 14913.041} C_VEL
LIN {X 0,Y 309.649,Z 599.18,A -85,B 0,C 180,E1 14913.978,E2 14913.978} C_VEL
LIN {X 0,Y 308.766,Z 647.995,A -85,B 0,C 180,E1 14915.633,E2 14915.633} C_VEL
LIN {X 0,Y 307.715,Z 675.867,A -85,B 0,C 180,E1 14917.684,E2 14917.684} C_VEL
LIN {X 0,Y 306.094,Z 700.85,A -85,B 0,C 180,E1 14920.743,E2 14920.743} C_VEL
LIN {X 0,Y 304.58,Z 720.79,A -85,B 0,C 180,E1 14924.51,E2 14924.51} C_VEL
LIN {X 0,Y 303.677,Z 734.739,A -85,B 0,C 180,E1 14928.528,E2 14928.528} C_VEL
LIN {X 0,Y 303.411,Z 743.915,A -85,B 0,C 180,E1 14932.852,E2 14932.852} C_VEL
LIN {X 0,Y 303.735,Z 748.136,A -85,B 0,C 180,E1 14937.146,E2 14937.146} C_VEL
LIN {X 0,Y 304.398,Z 748.373,A -85,B 0,C 180,E1 14939.994,E2 14939.994} C_VEL
LIN {X 0,Y 305.997,Z 744.847,A -85,B 0,C 180,E1 14944.236,E2 14944.236} C_VEL
LIN {X 0,Y 308.612,Z 735.263,A -85,B 0,C 180,E1 14948.783,E2 14948.783} C_VEL
LIN {X 0,Y 311.53,Z 721.2,A -85,B 0,C 180,E1 14952.584,E2 14952.584} C_VEL
LIN {X 0,Y 314.6,Z 701.268,A -85,B 0,C 180,E1 14955.999,E2 14955.999} C_VEL
LIN {X 0,Y 317.092,Z 676.553,A -85,B 0,C 180,E1 14958.659,E2 14958.659} C_VEL
LIN {X 0,Y 318.326,Z 648.709,A -85,B 0,C 180,E1 14960.365,E2 14960.365} C_VEL
LIN {X 0,Y 320.398,Z 598.127,A -85,B 0,C 180,E1 14962.334,E2 14962.334} C_VEL
LIN {X 0,Y 313.447,Z 578.373,A -85,B 0,C 180,E1 14964.552,E2 14964.552} C_VEL
LIN {X 0,Y 313.111,Z 576.079,A -85,B 0,C 180,E1 14965.011,E2 14965.011} C_VEL
LIN {X 0,Y 315.738,Z 576.618,A -85,B 0,C 180,E1 14965.945,E2 14965.945} C_VEL
LIN {X 0,Y 330.225,Z 601.581,A -85,B 0,C 180,E1 14972.178,E2 14972.178} C_VEL
LIN {X 0,Y 342.609,Z 627.099,A -85,B 0,C 180,E1 14976.99,E2 14976.99} C_VEL
LIN {X 0,Y 349.954,Z 647.257,A -85,B 0,C 180,E1 14980.072,E2 14980.072} C_VEL
LIN {X 0,Y 350.755,Z 657.292,A -85,B 0,C 180,E1 14981.117,E2 14981.117} C_VEL
LIN {X 0,Y 341.02,Z 700.949,A -85,B 0,C 180,E1 14984.299,E2 14984.299} C_VEL
LIN {X 0,Y 332.42,Z 733.558,A -85,B 0,C 180,E1 14987.642,E2 14987.642} C_VEL
LIN {X 0,Y 322.808,Z 764.323,A -85,B 0,C 180,E1 14992.148,E2 14992.148} C_VEL
LIN {X 0,Y 313.889,Z 790.969,A -85,B 0,C 180,E1 14997.698,E2 14997.698} C_VEL
LIN {X 0,Y 306.643,Z 813.077,A -85,B 0,C 180,E1 15004.245,E2 15004.245} C_VEL
LIN {X 0,Y 302.46,Z 828.296,A -85,B 0,C 180,E1 15010.712,E2 15010.712} C_VEL
LIN {X 0,Y 300.657,Z 838.24,A -85,B 0,C 180,E1 15016.945,E2 15016.945} C_VEL
LIN {X 0,Y 300.219,Z 842.86,A -85,B 0,C 180,E1 15021.326,E2 15021.326} C_VEL
LIN {X 0,Y 300.126,Z 846.011,A -85,B 0,C 180,E1 15027.117,E2 15027.117} C_VEL
LIN {X 0,Y 300.441,Z 846.423,A -85,B 0,C 180,E1 15029.999,E2 15029.999} C_VEL
LIN {X 0,Y 300.155,Z 843.742,A -85,B 0,C 180,E1 15037.221,E2 15037.221} C_VEL
LIN {X 0,Y 301.004,Z 835.789,A -85,B 0,C 180,E1 15044.518,E2 15044.518} C_VEL
LIN {X 0,Y 303.386,Z 823.588,A -85,B 0,C 180,E1 15051.139,E2 15051.139} C_VEL
LIN {X 0,Y 308.6,Z 804.872,A -85,B 0,C 180,E1 15057.989,E2 15057.989} C_VEL
LIN {X 0,Y 316.175,Z 781.069,A -85,B 0,C 180,E1 15064.048,E2 15064.048} C_VEL
LIN {X 0,Y 320.852,Z 766.162,A -85,B 0,C 180,E1 15066.966,E2 15066.966} C_VEL
LIN {X 0,Y 320.947,Z 754.379,A -85,B 0,C 180,E1 15069.286,E2 15069.286} C_VEL
LIN {X 0,Y 321.381,Z 741.931,A -85,B 0,C 180,E1 15071.481,E2 15071.481} C_VEL
LIN {X 0,Y 330.165,Z 709.711,A -85,B 0,C 180,E1 15075.176,E2 15075.176} C_VEL
LIN {X 0,Y 340.049,Z 666.379,A -85,B 0,C 180,E1 15078.618,E2 15078.618} C_VEL
LIN {X 0,Y 341.853,Z 653.26,A -85,B 0,C 180,E1 15079.566,E2 15079.566} C_VEL
LIN {X 0,Y 333.456,Z 627.955,A -85,B 0,C 180,E1 15083.165,E2 15083.165} C_VEL
LIN {X 0,Y 329.694,Z 621.045,A -85,B 0,C 180,E1 15084.445,E2 15084.445} C_VEL
LIN {X 0,Y 323.079,Z 631.478,A -85,B 0,C 180,E1 15084.839,E2 15084.839} C_VEL
LIN {X 0,Y 320.03,Z 634.578,A -85,B 0,C 180,E1 15085.275,E2 15085.275} C_VEL
LIN {X 0,Y 317.348,Z 666.2,A -85,B 0,C 180,E1 15087.334,E2 15087.334} C_VEL
LIN {X 0,Y 313.471,Z 693.614,A -85,B 0,C 180,E1 15090.246,E2 15090.246} C_VEL
LIN {X 0,Y 308.917,Z 716.287,A -85,B 0,C 180,E1 15093.926,E2 15093.926} C_VEL
LIN {X 0,Y 304.582,Z 733.214,A -85,B 0,C 180,E1 15098.194,E2 15098.194} C_VEL
LIN {X 0,Y 301.069,Z 743.802,A -85,B 0,C 180,E1 15102.505,E2 15102.505} C_VEL
LIN {X 0,Y 298.483,Z 749.521,A -85,B 0,C 180,E1 15106.857,E2 15106.857} C_VEL
LIN {X 0,Y 296.641,Z 751.01,A -85,B 0,C 180,E1 15111.228,E2 15111.228} C_VEL
LIN {X 0,Y 295.764,Z 748.427,A -85,B 0,C 180,E1 15115.617,E2 15115.617} C_VEL
LIN {X 0,Y 295.611,Z 740.401,A -85,B 0,C 180,E1 15120.738,E2 15120.738} C_VEL
LIN {X 0,Y 296.325,Z 726.146,A -85,B 0,C 180,E1 15125.852,E2 15125.852} C_VEL
LIN {X 0,Y 297.796,Z 707.658,A -85,B 0,C 180,E1 15130.223,E2 15130.223} C_VEL
LIN {X 0,Y 299.869,Z 682.904,A -85,B 0,C 180,E1 15134.208,E2 15134.208} C_VEL
LIN {X 0,Y 301.886,Z 654.069,A -85,B 0,C 180,E1 15137.272,E2 15137.272} C_VEL
LIN {X 0,Y 303.348,Z 621.657,A -85,B 0,C 180,E1 15139.333,E2 15139.333} C_VEL
LIN {X 0,Y 303.017,Z 597.498,A -85,B 0,C 180,E1 15140.239,E2 15140.239} C_VEL
LIN {X 0,Y 290.309,Z 549.53,A -85,B 0,C 180,E1 15142.692,E2 15142.692} C_VEL
LIN {X 0,Y 289.791,Z 549.813,A -85,B 0,C 180,E1 15148.572,E2 15148.572} C_VEL
LIN {X 0,Y 292.015,Z 555.001,A -85,B 0,C 180,E1 15150.129,E2 15150.129} C_VEL
LIN {X 0,Y 294.66,Z 558.31,A -85,B 0,C 180,E1 15151.564,E2 15151.564} C_VEL
LIN {X 0,Y 303.117,Z 571.579,A -85,B 0,C 180,E1 15155.808,E2 15155.808} C_VEL
LIN {X 0,Y 316.336,Z 594.447,A -85,B 0,C 180,E1 15161.348,E2 15161.348} C_VEL
LIN {X 0,Y 328.687,Z 621.126,A -85,B 0,C 180,E1 15166.089,E2 15166.089} C_VEL
LIN {X 0,Y 335.538,Z 644.159,A -85,B 0,C 180,E1 15169.623,E2 15169.623} C_VEL
LIN {X 0,Y 327.99,Z 678.346,A -85,B 0,C 180,E1 15172.849,E2 15172.849} C_VEL
LIN {X 0,Y 318.807,Z 709.556,A -85,B 0,C 180,E1 15177.018,E2 15177.018} C_VEL
LIN {X 0,Y 310.08,Z 735.914,A -85,B 0,C 180,E1 15182.066,E2 15182.066} C_VEL
LIN {X 0,Y 302.266,Z 758.393,A -85,B 0,C 180,E1 15188.179,E2 15188.179} C_VEL
LIN {X 0,Y 296.718,Z 775.659,A -85,B 0,C 180,E1 15195.106,E2 15195.106} C_VEL
LIN {X 0,Y 294.16,Z 785.449,A -85,B 0,C 180,E1 15201.147,E2 15201.147} C_VEL
LIN {X 0,Y 293.119,Z 791.112,A -85,B 0,C 180,E1 15207.049,E2 15207.049} C_VEL
LIN {X 0,Y 292.755,Z 793.142,A -85,B 0,C 180,E1 15212.956,E2 15212.956} C_VEL
LIN {X 0,Y 293.236,Z 790.682,A -85,B 0,C 180,E1 15220.378,E2 15220.378} C_VEL
LIN {X 0,Y 295.378,Z 782.505,A -85,B 0,C 180,E1 15227.853,E2 15227.853} C_VEL
LIN {X 0,Y 299.581,Z 769.716,A -85,B 0,C 180,E1 15234.502,E2 15234.502} C_VEL
LIN {X 0,Y 306.756,Z 750.83,A -85,B 0,C 180,E1 15241.019,E2 15241.019} C_VEL
LIN {X 0,Y 315.791,Z 726.895,A -85,B 0,C 180,E1 15246.683,E2 15246.683} C_VEL
LIN {X 0,Y 325.106,Z 699.851,A -85,B 0,C 180,E1 15251.215,E2 15251.215} C_VEL
LIN {X 0,Y 334.656,Z 667.391,A -85,B 0,C 180,E1 15255.029,E2 15255.029} C_VEL
LIN {X 0,Y 339.426,Z 646.405,A -85,B 0,C 180,E1 15256.871,E2 15256.871} C_VEL
LIN {X 0,Y 331.272,Z 621.223,A -85,B 0,C 180,E1 15261.187,E2 15261.187} C_VEL
LIN {X 0,Y 319.496,Z 596.965,A -85,B 0,C 180,E1 15266.182,E2 15266.182} C_VEL
LIN {X 0,Y 309.518,Z 579.907,A -85,B 0,C 180,E1 15270.921,E2 15270.921} C_VEL
LIN {X 0,Y 305.583,Z 584.407,A -85,B 0,C 180,E1 15271.873,E2 15271.873} C_VEL
LIN {X 0,Y 301.925,Z 590.049,A -85,B 0,C 180,E1 15272.644,E2 15272.644} C_VEL
LIN {X 0,Y 300.629,Z 590.632,A -85,B 0,C 180,E1 15273.236,E2 15273.236} C_VEL
LIN {X 0,Y 301.908,Z 604.031,A -85,B 0,C 180,E1 15273.738,E2 15273.738} C_VEL
LIN {X 0,Y 301.031,Z 650.807,A -85,B 0,C 180,E1 15275.422,E2 15275.422} C_VEL
LIN {X 0,Y 299.9,Z 678.502,A -85,B 0,C 180,E1 15277.576,E2 15277.576} C_VEL
LIN {X 0,Y 298.197,Z 703.41,A -85,B 0,C 180,E1 15280.789,E2 15280.789} C_VEL
LIN {X 0,Y 296.704,Z 722.924,A -85,B 0,C 180,E1 15284.65,E2 15284.65} C_VEL
LIN {X 0,Y 295.792,Z 737.144,A -85,B 0,C 180,E1 15288.964,E2 15288.964} C_VEL
LIN {X 0,Y 295.622,Z 745.898,A -85,B 0,C 180,E1 15293.398,E2 15293.398} C_VEL
LIN {X 0,Y 295.939,Z 749.42,A -85,B 0,C 180,E1 15297.07,E2 15297.07} C_VEL
LIN {X 0,Y 296.648,Z 749.921,A -85,B 0,C 180,E1 15299.993,E2 15299.993} C_VEL
LIN {X 0,Y 298.708,Z 745.798,A -85,B 0,C 180,E1 15305.065,E2 15305.065} C_VEL
LIN {X 0,Y 301.669,Z 735.663,A -85,B 0,C 180,E1 15309.713,E2 15309.713} C_VEL
LIN {X 0,Y 304.908,Z 720.97,A -85,B 0,C 180,E1 15313.59,E2 15313.59} C_VEL
LIN {X 0,Y 308.234,Z 700.139,A -85,B 0,C 180,E1 15317.075,E2 15317.075} C_VEL
LIN {X 0,Y 310.93,Z 673.921,A -85,B 0,C 180,E1 15319.761,E2 15319.761} C_VEL
LIN {X 0,Y 312.114,Z 646.299,A -85,B 0,C 180,E1 15321.347,E2 15321.347} C_VEL
LIN {X 0,Y 314.363,Z 600.123,A -85,B 0,C 180,E1 15323.224,E2 15323.224} C_VEL
LIN {X 0,Y 310.076,Z 586.11,A -85,B 0,C 180,E1 15324.939,E2 15324.939} C_VEL
LIN {X 0,Y 312.887,Z 584.288,A -85,B 0,C 180,E1 15325.719,E2 15325.719} C_VEL
LIN {X 0,Y 326.337,Z 608.168,A -85,B 0,C 180,E1 15331.785,E2 15331.785} C_VEL
LIN {X 0,Y 338.055,Z 633.493,A -85,B 0,C 180,E1 15336.66,E2 15336.66} C_VEL
LIN {X 0,Y 344.461,Z 653.112,A -85,B 0,C 180,E1 15339.673,E2 15339.673} C_VEL
LIN {X 0,Y 344.46,Z 660.428,A -85,B 0,C 180,E1 15340.39,E2 15340.39} C_VEL
LIN {X 0,Y 334.133,Z 704.717,A -85,B 0,C 180,E1 15343.724,E2 15343.724} C_VEL
LIN {X 0,Y 325.151,Z 736.814,A -85,B 0,C 180,E1 15347.208,E2 15347.208} C_VEL
LIN {X 0,Y 315.193,Z 766.67,A -85,B 0,C 180,E1 15351.817,E2 15351.817} C_VEL
LIN {X 0,Y 305.971,Z 792.834,A -85,B 0,C 180,E1 15357.56,E2 15357.56} C_VEL
LIN {X 0,Y 299.057,Z 812.973,A -85,B 0,C 180,E1 15363.796,E2 15363.796} C_VEL
LIN {X 0,Y 294.36,Z 829.272,A -85,B 0,C 180,E1 15371.121,E2 15371.121} C_VEL
LIN {X 0,Y 292.551,Z 839.722,A -85,B 0,C 180,E1 15378.503,E2 15378.503} C_VEL
LIN {X 0,Y 292.17,Z 844.137,A -85,B 0,C 180,E1 15384.07,E2 15384.07} C_VEL
LIN {X 0,Y 292.588,Z 845.715,A -85,B 0,C 180,E1 15389.999,E2 15389.999} C_VEL
LIN {X 0,Y 292.303,Z 843.002,A -85,B 0,C 180,E1 15397.416,E2 15397.416} C_VEL
LIN {X 0,Y 293.226,Z 834.99,A -85,B 0,C 180,E1 15404.912,E2 15404.912} C_VEL
LIN {X 0,Y 295.75,Z 822.705,A -85,B 0,C 180,E1 15411.712,E2 15411.712} C_VEL
LIN {X 0,Y 301.224,Z 804.325,A -85,B 0,C 180,E1 15418.592,E2 15418.592} C_VEL
LIN {X 0,Y 308.882,Z 781.198,A -85,B 0,C 180,E1 15424.633,E2 15424.633} C_VEL
LIN {X 0,Y 317.944,Z 753.226,A -85,B 0,C 180,E1 15429.832,E2 15429.832} C_VEL
LIN {X 0,Y 321.381,Z 741.931,A -85,B 0,C 180,E1 15431.481,E2 15431.481} C_VEL
LIN {X 0,Y 322.021,Z 728.842,A -85,B 0,C 180,E1 15433.551,E2 15433.551} C_VEL
LIN {X 0,Y 322.544,Z 715.14,A -85,B 0,C 180,E1 15435.505,E2 15435.505} C_VEL
LIN {X 0,Y 332.816,Z 672.601,A -85,B 0,C 180,E1 15439.093,E2 15439.093} C_VEL
LIN {X 0,Y 335.733,Z 655.945,A -85,B 0,C 180,E1 15440.294,E2 15440.294} C_VEL
LIN {X 0,Y 328.086,Z 633.638,A -85,B 0,C 180,E1 15443.67,E2 15443.67} C_VEL
LIN {X 0,Y 321.488,Z 641.563,A -85,B 0,C 180,E1 15444.199,E2 15444.199} C_VEL
LIN {X 0,Y 316.159,Z 647.94,A -85,B 0,C 180,E1 15444.621,E2 15444.621} C_VEL
LIN {X 0,Y 313.887,Z 649.673,A -85,B 0,C 180,E1 15444.97,E2 15444.97} C_VEL
LIN {X 0,Y 310.134,Z 680.163,A -85,B 0,C 180,E1 15447.505,E2 15447.505} C_VEL
LIN {X 0,Y 305.477,Z 705.458,A -85,B 0,C 180,E1 15450.81,E2 15450.81} C_VEL
LIN {X 0,Y 300.601,Z 725.452,A -85,B 0,C 180,E1 15454.784,E2 15454.784} C_VEL
LIN {X 0,Y 296.197,Z 739.526,A -85,B 0,C 180,E1 15459.114,E2 15459.114} C_VEL
LIN {X 0,Y 292.67,Z 748.278,A -85,B 0,C 180,E1 15463.654,E2 15463.654} C_VEL
LIN {X 0,Y 290.185,Z 752.139,A -85,B 0,C 180,E1 15468.001,E2 15468.001} C_VEL
LIN {X 0,Y 288.98,Z 752.578,A -85,B 0,C 180,E1 15470.994,E2 15470.994} C_VEL
LIN {X 0,Y 287.997,Z 749.762,A -85,B 0,C 180,E1 15475.519,E2 15475.519} C_VEL
LIN {X 0,Y 287.772,Z 741.48,A -85,B 0,C 180,E1 15480.758,E2 15480.758} C_VEL
LIN {X 0,Y 288.525,Z 726.942,A -85,B 0,C 180,E1 15486.011,E2 15486.011} C_VEL
LIN {X 0,Y 290.048,Z 708.018,A -85,B 0,C 180,E1 15490.499,E2 15490.499} C_VEL
LIN {X 0,Y 292.093,Z 684.125,A -85,B 0,C 180,E1 15494.403,E2 15494.403} C_VEL
LIN {X 0,Y 294.155,Z 655.328,A -85,B 0,C 180,E1 15497.548,E2 15497.548} C_VEL
LIN {X 0,Y 295.71,Z 622.859,A -85,B 0,C 180,E1 15499.675,E2 15499.675} C_VEL
LIN {X 0,Y 295.386,Z 598.701,A -85,B 0,C 180,E1 15500.609,E2 15500.609} C_VEL
LIN {X 0,Y 282.298,Z 549.53,A -85,B 0,C 180,E1 15503.333,E2 15503.333} C_VEL
LIN {X 0,Y 282.168,Z 550.375,A -85,B 0,C 180,E1 15504.748,E2 15504.748} C_VEL
LIN {X 0,Y 284.745,Z 555.555,A -85,B 0,C 180,E1 15506.852,E2 15506.852} C_VEL
LIN {X 0,Y 286.959,Z 558.142,A -85,B 0,C 180,E1 15508.255,E2 15508.255} C_VEL
LIN {X 0,Y 295.758,Z 571.826,A -85,B 0,C 180,E1 15513.363,E2 15513.363} C_VEL
LIN {X 0,Y 307.692,Z 592.203,A -85,B 0,C 180,E1 15518.968,E2 15518.968} C_VEL
LIN {X 0,Y 319.48,Z 615.847,A -85,B 0,C 180,E1 15523.736,E2 15523.736} C_VEL
LIN {X 0,Y 328.36,Z 642.358,A -85,B 0,C 180,E1 15528.133,E2 15528.133} C_VEL
LIN {X 0,Y 329.355,Z 649.532,A -85,B 0,C 180,E1 15529.139,E2 15529.139} C_VEL
LIN {X 0,Y 320.722,Z 683.42,A -85,B 0,C 180,E1 15532.459,E2 15532.459} C_VEL
LIN {X 0,Y 311.598,Z 712.593,A -85,B 0,C 180,E1 15536.57,E2 15536.57} C_VEL
LIN {X 0,Y 302.606,Z 738.426,A -85,B 0,C 180,E1 15541.72,E2 15541.72} C_VEL
LIN {X 0,Y 294.846,Z 759.609,A -85,B 0,C 180,E1 15547.719,E2 15547.719} C_VEL
LIN {X 0,Y 288.995,Z 776.782,A -85,B 0,C 180,E1 15554.865,E2 15554.865} C_VEL
LIN {X 0,Y 286.382,Z 786.227,A -85,B 0,C 180,E1 15560.904,E2 15560.904} C_VEL
LIN {X 0,Y 285.271,Z 791.851,A -85,B 0,C 180,E1 15566.968,E2 15566.968} C_VEL
LIN {X 0,Y 284.876,Z 793.856,A -85,B 0,C 180,E1 15573.037,E2 15573.037} C_VEL
LIN {X 0,Y 285.436,Z 791.36,A -85,B 0,C 180,E1 15580.665,E2 15580.665} C_VEL
LIN {X 0,Y 287.769,Z 783.164,A -85,B 0,C 180,E1 15588.341,E2 15588.341} C_VEL
LIN {X 0,Y 292.293,Z 770.35,A -85,B 0,C 180,E1 15595.155,E2 15595.155} C_VEL
LIN {X 0,Y 299.99,Z 751.173,A -85,B 0,C 180,E1 15601.885,E2 15601.885} C_VEL
LIN {X 0,Y 309.408,Z 727.483,A -85,B 0,C 180,E1 15607.569,E2 15607.569} C_VEL
LIN {X 0,Y 319.467,Z 699.51,A -85,B 0,C 180,E1 15612.285,E2 15612.285} C_VEL
LIN {X 0,Y 329.079,Z 667.857,A -85,B 0,C 180,E1 15616.009,E2 15616.009} C_VEL
LIN {X 0,Y 333.466,Z 649.295,A -85,B 0,C 180,E1 15617.682,E2 15617.682} C_VEL
LIN {X 0,Y 325.873,Z 624.977,A -85,B 0,C 180,E1 15622.061,E2 15622.061} C_VEL
LIN {X 0,Y 314.22,Z 600.359,A -85,B 0,C 180,E1 15627.392,E2 15627.392} C_VEL
LIN {X 0,Y 307.461,Z 589.042,A -85,B 0,C 180,E1 15630.7,E2 15630.7} C_VEL
LIN {X 0,Y 302.203,Z 596.534,A -85,B 0,C 180,E1 15631.775,E2 15631.775} C_VEL
LIN {X 0,Y 299.077,Z 602.507,A -85,B 0,C 180,E1 15632.273,E2 15632.273} C_VEL
LIN {X 0,Y 295.311,Z 608.472,A -85,B 0,C 180,E1 15633.014,E2 15633.014} C_VEL
LIN {X 0,Y 294.202,Z 609.361,A -85,B 0,C 180,E1 15633.508,E2 15633.508} C_VEL
LIN {X 0,Y 293.34,Z 652.239,A -85,B 0,C 180,E1 15635.14,E2 15635.14} C_VEL
LIN {X 0,Y 292.148,Z 680.233,A -85,B 0,C 180,E1 15637.401,E2 15637.401} C_VEL
LIN {X 0,Y 290.384,Z 704.878,A -85,B 0,C 180,E1 15640.672,E2 15640.672} C_VEL
LIN {X 0,Y 288.914,Z 723.718,A -85,B 0,C 180,E1 15644.466,E2 15644.466} C_VEL
LIN {X 0,Y 288.002,Z 737.585,A -85,B 0,C 180,E1 15648.661,E2 15648.661} C_VEL
LIN {X 0,Y 287.824,Z 746.79,A -85,B 0,C 180,E1 15653.218,E2 15653.218} C_VEL
LIN {X 0,Y 288.165,Z 750.68,A -85,B 0,C 180,E1 15656.991,E2 15656.991} C_VEL
LIN {X 0,Y 288.897,Z 751.433,A -85,B 0,C 180,E1 15659.993,E2 15659.993} C_VEL
LIN {X 0,Y 291.093,Z 747.768,A -85,B 0,C 180,E1 15665.198,E2 15665.198} C_VEL
LIN {X 0,Y 293.969,Z 739.15,A -85,B 0,C 180,E1 15669.597,E2 15669.597} C_VEL
LIN {X 0,Y 297.697,Z 724.109,A -85,B 0,C 180,E1 15673.926,E2 15673.926} C_VEL
LIN {X 0,Y 301.277,Z 704.216,A -85,B 0,C 180,E1 15677.482,E2 15677.482} C_VEL
LIN {X 0,Y 304.122,Z 680.934,A -85,B 0,C 180,E1 15680.128,E2 15680.128} C_VEL
LIN {X 0,Y 305.807,Z 653.821,A -85,B 0,C 180,E1 15681.965,E2 15681.965} C_VEL
LIN {X 0,Y 308.497,Z 602.047,A -85,B 0,C 180,E1 15684.198,E2 15684.198} C_VEL
LIN {X 0,Y 307.227,Z 596.038,A -85,B 0,C 180,E1 15685,E2 15685} C_VEL
LIN {X 0,Y 310.724,Z 593.369,A -85,B 0,C 180,E1 15685.911,E2 15685.911} C_VEL
LIN {X 0,Y 323.586,Z 616.954,A -85,B 0,C 180,E1 15691.915,E2 15691.915} C_VEL
LIN {X 0,Y 335.377,Z 645.011,A -85,B 0,C 180,E1 15697.216,E2 15697.216} C_VEL
LIN {X 0,Y 338.918,Z 658.881,A -85,B 0,C 180,E1 15699.269,E2 15699.269} C_VEL
LIN {X 0,Y 327.862,Z 706.119,A -85,B 0,C 180,E1 15702.929,E2 15702.929} C_VEL
LIN {X 0,Y 318.309,Z 738.531,A -85,B 0,C 180,E1 15706.568,E2 15706.568} C_VEL
LIN {X 0,Y 307.832,Z 768.35,A -85,B 0,C 180,E1 15711.35,E2 15711.35} C_VEL
LIN {X 0,Y 298.514,Z 793.386,A -85,B 0,C 180,E1 15717.078,E2 15717.078} C_VEL
LIN {X 0,Y 290.985,Z 814.15,A -85,B 0,C 180,E1 15723.841,E2 15723.841} C_VEL
LIN {X 0,Y 286.289,Z 830.213,A -85,B 0,C 180,E1 15731.561,E2 15731.561} C_VEL
LIN {X 0,Y 284.74,Z 838.568,A -85,B 0,C 180,E1 15737.759,E2 15737.759} C_VEL
LIN {X 0,Y 284.28,Z 843.436,A -85,B 0,C 180,E1 15743.905,E2 15743.905} C_VEL
LIN {X 0,Y 284.709,Z 845.005,A -85,B 0,C 180,E1 15749.999,E2 15749.999} C_VEL
LIN {X 0,Y 284.419,Z 842.258,A -85,B 0,C 180,E1 15757.622,E2 15757.622} C_VEL
LIN {X 0,Y 285.409,Z 834.183,A -85,B 0,C 180,E1 15765.33,E2 15765.33} C_VEL
LIN {X 0,Y 288.593,Z 820.34,A -85,B 0,C 180,E1 15772.997,E2 15772.997} C_VEL
LIN {X 0,Y 294.987,Z 800.309,A -85,B 0,C 180,E1 15780.289,E2 15780.289} C_VEL
LIN {X 0,Y 303.163,Z 776.87,A -85,B 0,C 180,E1 15786.238,E2 15786.238} C_VEL
LIN {X 0,Y 312.68,Z 748.467,A -85,B 0,C 180,E1 15791.34,E2 15791.34} C_VEL
LIN {X 0,Y 322.281,Z 716.188,A -85,B 0,C 180,E1 15795.393,E2 15795.393} C_VEL
LIN {X 0,Y 322.544,Z 715.14,A -85,B 0,C 180,E1 15795.505,E2 15795.505} C_VEL
LIN {X 0,Y 323.045,Z 700.916,A -85,B 0,C 180,E1 15797.339,E2 15797.339} C_VEL
LIN {X 0,Y 323.743,Z 686.215,A -85,B 0,C 180,E1 15799.014,E2 15799.014} C_VEL
LIN {X 0,Y 329.714,Z 659.304,A -85,B 0,C 180,E1 15800.959,E2 15800.959} C_VEL
LIN {X 0,Y 325.71,Z 645.908,A -85,B 0,C 180,E1 15802.973,E2 15802.973} C_VEL
LIN {X 0,Y 323.363,Z 647.783,A -85,B 0,C 180,E1 15803.232,E2 15803.232} C_VEL
LIN {X 0,Y 310.363,Z 661.291,A -85,B 0,C 180,E1 15804.314,E2 15804.314} C_VEL
LIN {X 0,Y 307.631,Z 663.534,A -85,B 0,C 180,E1 15804.75,E2 15804.75} C_VEL
LIN {X 0,Y 302.972,Z 691.765,A -85,B 0,C 180,E1 15807.619,E2 15807.619} C_VEL
LIN {X 0,Y 297.673,Z 714.907,A -85,B 0,C 180,E1 15811.218,E2 15811.218} C_VEL
LIN {X 0,Y 292.259,Z 733.314,A -85,B 0,C 180,E1 15815.61,E2 15815.61} C_VEL
LIN {X 0,Y 287.736,Z 745.093,A -85,B 0,C 180,E1 15820.078,E2 15820.078} C_VEL
LIN {X 0,Y 284.373,Z 751.812,A -85,B 0,C 180,E1 15824.621,E2 15824.621} C_VEL
LIN {X 0,Y 282.634,Z 753.852,A -85,B 0,C 180,E1 15827.676,E2 15827.676} C_VEL
LIN {X 0,Y 281.305,Z 754.134,A -85,B 0,C 180,E1 15830.746,E2 15830.746} C_VEL
LIN {X 0,Y 280.233,Z 751.093,A -85,B 0,C 180,E1 15835.394,E2 15835.394} C_VEL
LIN {X 0,Y 279.945,Z 742.516,A -85,B 0,C 180,E1 15840.779,E2 15840.779} C_VEL
LIN {X 0,Y 280.706,Z 727.651,A -85,B 0,C 180,E1 15846.179,E2 15846.179} C_VEL
LIN {X 0,Y 282.44,Z 706.449,A -85,B 0,C 180,E1 15851.175,E2 15851.175} C_VEL
LIN {X 0,Y 284.677,Z 681.027,A -85,B 0,C 180,E1 15855.18,E2 15855.18} C_VEL
LIN {X 0,Y 286.798,Z 650.761,A -85,B 0,C 180,E1 15858.311,E2 15858.311} C_VEL
LIN {X 0,Y 288.216,Z 618.239,A -85,B 0,C 180,E1 15860.268,E2 15860.268} C_VEL
LIN {X 0,Y 287.681,Z 599.731,A -85,B 0,C 180,E1 15860.996,E2 15860.996} C_VEL
LIN {X 0,Y 277.251,Z 559.833,A -85,B 0,C 180,E1 15863.231,E2 15863.231} C_VEL
LIN {X 0,Y 279.437,Z 557.887,A -85,B 0,C 180,E1 15864.268,E2 15864.268} C_VEL
LIN {X 0,Y 282.907,Z 563.41,A -85,B 0,C 180,E1 15866.969,E2 15866.969} C_VEL
LIN {X 0,Y 292.401,Z 578.498,A -85,B 0,C 180,E1 15872.848,E2 15872.848} C_VEL
LIN {X 0,Y 304.399,Z 599.46,A -85,B 0,C 180,E1 15878.704,E2 15878.704} C_VEL
LIN {X 0,Y 316.077,Z 624.781,A -85,B 0,C 180,E1 15883.82,E2 15883.82} C_VEL
LIN {X 0,Y 323.419,Z 650.385,A -85,B 0,C 180,E1 15888.155,E2 15888.155} C_VEL
LIN {X 0,Y 314.922,Z 683.5,A -85,B 0,C 180,E1 15891.466,E2 15891.466} C_VEL
LIN {X 0,Y 305.086,Z 713.659,A -85,B 0,C 180,E1 15895.759,E2 15895.759} C_VEL
LIN {X 0,Y 295.703,Z 739.397,A -85,B 0,C 180,E1 15900.998,E2 15900.998} C_VEL
LIN {X 0,Y 287.336,Z 761.114,A -85,B 0,C 180,E1 15907.339,E2 15907.339} C_VEL
LIN {X 0,Y 281.388,Z 777.604,A -85,B 0,C 180,E1 15914.445,E2 15914.445} C_VEL
LIN {X 0,Y 278.621,Z 787.004,A -85,B 0,C 180,E1 15920.649,E2 15920.649} C_VEL
LIN {X 0,Y 277.429,Z 792.588,A -85,B 0,C 180,E1 15926.882,E2 15926.882} C_VEL
LIN {X 0,Y 277.018,Z 794.567,A -85,B 0,C 180,E1 15933.124,E2 15933.124} C_VEL
LIN {X 0,Y 277.361,Z 792.997,A -85,B 0,C 180,E1 15939.395,E2 15939.395} C_VEL
LIN {X 0,Y 278.842,Z 787.802,A -85,B 0,C 180,E1 15945.701,E2 15945.701} C_VEL
LIN {X 0,Y 282.636,Z 777.327,A -85,B 0,C 180,E1 15952.776,E2 15952.776} C_VEL
LIN {X 0,Y 289.224,Z 761.175,A -85,B 0,C 180,E1 15959.686,E2 15959.686} C_VEL
LIN {X 0,Y 298.523,Z 739.313,A -85,B 0,C 180,E1 15966.01,E2 15966.01} C_VEL
LIN {X 0,Y 309.257,Z 712.073,A -85,B 0,C 180,E1 15971.442,E2 15971.442} C_VEL
LIN {X 0,Y 319.958,Z 680.74,A -85,B 0,C 180,E1 15975.726,E2 15975.726} C_VEL
LIN {X 0,Y 327.513,Z 652.12,A -85,B 0,C 180,E1 15978.546,E2 15978.546} C_VEL
LIN {X 0,Y 320.306,Z 628.145,A -85,B 0,C 180,E1 15983.074,E2 15983.074} C_VEL
LIN {X 0,Y 309.474,Z 605.023,A -85,B 0,C 180,E1 15988.379,E2 15988.379} C_VEL
LIN {X 0,Y 305.986,Z 599.124,A -85,B 0,C 180,E1 15990.138,E2 15990.138} C_VEL
LIN {X 0,Y 302.074,Z 604.561,A -85,B 0,C 180,E1 15990.915,E2 15990.915} C_VEL
LIN {X 0,Y 296.352,Z 614.068,A -85,B 0,C 180,E1 15991.897,E2 15991.897} C_VEL
LIN {X 0,Y 294.627,Z 616.975,A -85,B 0,C 180,E1 15992.2,E2 15992.2} C_VEL
LIN {X 0,Y 289.221,Z 628.007,A -85,B 0,C 180,E1 15992.833,E2 15992.833} C_VEL
LIN {X 0,Y 286.338,Z 630.39,A -85,B 0,C 180,E1 15993.67,E2 15993.67} C_VEL
LIN {X 0,Y 285.074,Z 666.718,A -85,B 0,C 180,E1 15995.772,E2 15995.772} C_VEL
LIN {X 0,Y 283.593,Z 693.621,A -85,B 0,C 180,E1 15998.628,E2 15998.628} C_VEL
LIN {X 0,Y 281.67,Z 716.49,A -85,B 0,C 180,E1 16002.454,E2 16002.454} C_VEL
LIN {X 0,Y 280.476,Z 734.061,A -85,B 0,C 180,E1 16007.003,E2 16007.003} C_VEL
LIN {X 0,Y 279.981,Z 745.002,A -85,B 0,C 180,E1 16011.469,E2 16011.469} C_VEL
LIN {X 0,Y 280.165,Z 750.661,A -85,B 0,C 180,E1 16015.447,E2 16015.447} C_VEL
LIN {X 0,Y 281.122,Z 752.915,A -85,B 0,C 180,E1 16019.993,E2 16019.993} C_VEL
LIN {X 0,Y 283.054,Z 750.614,A -85,B 0,C 180,E1 16024.58,E2 16024.58} C_VEL
LIN {X 0,Y 285.93,Z 743.375,A -85,B 0,C 180,E1 16029.103,E2 16029.103} C_VEL
LIN {X 0,Y 289.753,Z 730.238,A -85,B 0,C 180,E1 16033.547,E2 16033.547} C_VEL
LIN {X 0,Y 293.779,Z 711.558,A -85,B 0,C 180,E1 16037.411,E2 16037.411} C_VEL
LIN {X 0,Y 297.449,Z 687.246,A -85,B 0,C 180,E1 16040.552,E2 16040.552} C_VEL
LIN {X 0,Y 299.627,Z 659.532,A -85,B 0,C 180,E1 16042.674,E2 16042.674} C_VEL
LIN {X 0,Y 303.747,Z 607.041,A -85,B 0,C 180,E1 16045.054,E2 16045.054} C_VEL
LIN {X 0,Y 308.516,Z 602.077,A -85,B 0,C 180,E1 16046.11,E2 16046.11} C_VEL
LIN {X 0,Y 321.515,Z 627.979,A -85,B 0,C 180,E1 16052.5,E2 16052.5} C_VEL
LIN {X 0,Y 331.902,Z 655.481,A -85,B 0,C 180,E1 16057.608,E2 16057.608} C_VEL
LIN {X 0,Y 332.884,Z 663.278,A -85,B 0,C 180,E1 16058.62,E2 16058.62} C_VEL
LIN {X 0,Y 321.507,Z 708.07,A -85,B 0,C 180,E1 16062.149,E2 16062.149} C_VEL
LIN {X 0,Y 311.573,Z 740.062,A -85,B 0,C 180,E1 16065.869,E2 16065.869} C_VEL
LIN {X 0,Y 300.889,Z 768.858,A -85,B 0,C 180,E1 16070.643,E2 16070.643} C_VEL
LIN {X 0,Y 290.948,Z 794.26,A -85,B 0,C 180,E1 16076.674,E2 16076.674} C_VEL
LIN {X 0,Y 282.957,Z 815.334,A -85,B 0,C 180,E1 16083.894,E2 16083.894} C_VEL
LIN {X 0,Y 278.252,Z 830.8,A -85,B 0,C 180,E1 16091.889,E2 16091.889} C_VEL
LIN {X 0,Y 276.705,Z 839.376,A -85,B 0,C 180,E1 16098.966,E2 16098.966} C_VEL
LIN {X 0,Y 276.474,Z 843.9,A -85,B 0,C 180,E1 16106.87,E2 16106.87} C_VEL
LIN {X 0,Y 276.855,Z 844.297,A -85,B 0,C 180,E1 16109.999,E2 16109.999} C_VEL
LIN {X 0,Y 276.535,Z 841.512,A -85,B 0,C 180,E1 16117.841,E2 16117.841} C_VEL
LIN {X 0,Y 277.606,Z 833.373,A -85,B 0,C 180,E1 16125.772,E2 16125.772} C_VEL
LIN {X 0,Y 281.183,Z 819.091,A -85,B 0,C 180,E1 16133.804,E2 16133.804} C_VEL
LIN {X 0,Y 287.958,Z 799.134,A -85,B 0,C 180,E1 16141.165,E2 16141.165} C_VEL
LIN {X 0,Y 296.551,Z 775.709,A -85,B 0,C 180,E1 16147.18,E2 16147.18} C_VEL
LIN {X 0,Y 306.71,Z 746.55,A -85,B 0,C 180,E1 16152.448,E2 16152.448} C_VEL
LIN {X 0,Y 316.52,Z 714.544,A -85,B 0,C 180,E1 16156.46,E2 16156.46} C_VEL
LIN {X 0,Y 323.743,Z 686.215,A -85,B 0,C 180,E1 16159.014,E2 16159.014} C_VEL
LIN {X 0,Y 324.913,Z 670.952,A -85,B 0,C 180,E1 16160.555,E2 16160.555} C_VEL
LIN {X 0,Y 322.221,Z 657.078,A -85,B 0,C 180,E1 16162.494,E2 16162.494} C_VEL
LIN {X 0,Y 303.137,Z 674.306,A -85,B 0,C 180,E1 16164.211,E2 16164.211} C_VEL
LIN {X 0,Y 301.184,Z 676.359,A -85,B 0,C 180,E1 16164.605,E2 16164.605} C_VEL
LIN {X 0,Y 295.708,Z 702.357,A -85,B 0,C 180,E1 16167.791,E2 16167.791} C_VEL
LIN {X 0,Y 289.762,Z 723.39,A -85,B 0,C 180,E1 16171.634,E2 16171.634} C_VEL
LIN {X 0,Y 284.166,Z 739.301,A -85,B 0,C 180,E1 16176.122,E2 16176.122} C_VEL
LIN {X 0,Y 279.297,Z 749.947,A -85,B 0,C 180,E1 16181.092,E2 16181.092} C_VEL
LIN {X 0,Y 276.966,Z 753.705,A -85,B 0,C 180,E1 16184.199,E2 16184.199} C_VEL
LIN {X 0,Y 275.074,Z 755.583,A -85,B 0,C 180,E1 16187.331,E2 16187.331} C_VEL
LIN {X 0,Y 273.627,Z 755.679,A -85,B 0,C 180,E1 16190.484,E2 16190.484} C_VEL
LIN {X 0,Y 272.328,Z 751.592,A -85,B 0,C 180,E1 16195.954,E2 16195.954} C_VEL
LIN {X 0,Y 272.141,Z 741.775,A -85,B 0,C 180,E1 16201.596,E2 16201.596} C_VEL
LIN {X 0,Y 273.143,Z 725.486,A -85,B 0,C 180,E1 16207.148,E2 16207.148} C_VEL
LIN {X 0,Y 274.995,Z 703.419,A -85,B 0,C 180,E1 16212.083,E2 16212.083} C_VEL
LIN {X 0,Y 277.441,Z 675.927,A -85,B 0,C 180,E1 16216.193,E2 16216.193} C_VEL
LIN {X 0,Y 279.523,Z 644.992,A -85,B 0,C 180,E1 16219.153,E2 16219.153} C_VEL
LIN {X 0,Y 280.717,Z 611.727,A -85,B 0,C 180,E1 16220.925,E2 16220.925} C_VEL
LIN {X 0,Y 279.696,Z 599.584,A -85,B 0,C 180,E1 16221.446,E2 16221.446} C_VEL
LIN {X 0,Y 273.15,Z 573.726,A -85,B 0,C 180,E1 16222.943,E2 16222.943} C_VEL
LIN {X 0,Y 275.762,Z 570.386,A -85,B 0,C 180,E1 16224.023,E2 16224.023} C_VEL
LIN {X 0,Y 277.452,Z 567.057,A -85,B 0,C 180,E1 16224.509,E2 16224.509} C_VEL
LIN {X 0,Y 281.575,Z 573.307,A -85,B 0,C 180,E1 16227.648,E2 16227.648} C_VEL
LIN {X 0,Y 289.093,Z 585.296,A -85,B 0,C 180,E1 16232.355,E2 16232.355} C_VEL
LIN {X 0,Y 300.488,Z 605.905,A -85,B 0,C 180,E1 16238.202,E2 16238.202} C_VEL
LIN {X 0,Y 310.961,Z 629.6,A -85,B 0,C 180,E1 16243.161,E2 16243.161} C_VEL
LIN {X 0,Y 317.436,Z 653.599,A -85,B 0,C 180,E1 16247.403,E2 16247.403} C_VEL
LIN {X 0,Y 307.968,Z 687.602,A -85,B 0,C 180,E1 16250.909,E2 16250.909} C_VEL
LIN {X 0,Y 297.94,Z 716.675,A -85,B 0,C 180,E1 16255.26,E2 16255.26} C_VEL
LIN {X 0,Y 287.642,Z 743.296,A -85,B 0,C 180,E1 16260.993,E2 16260.993} C_VEL
LIN {X 0,Y 278.961,Z 764.815,A -85,B 0,C 180,E1 16267.747,E2 16267.747} C_VEL
LIN {X 0,Y 273.02,Z 780.742,A -85,B 0,C 180,E1 16275.334,E2 16275.334} C_VEL
LIN {X 0,Y 270.387,Z 789.525,A -85,B 0,C 180,E1 16281.979,E2 16281.979} C_VEL
LIN {X 0,Y 269.588,Z 793.324,A -85,B 0,C 180,E1 16286.791,E2 16286.791} C_VEL
LIN {X 0,Y 269.165,Z 795.279,A -85,B 0,C 180,E1 16293.215,E2 16293.215} C_VEL
LIN {X 0,Y 269.716,Z 793.008,A -85,B 0,C 180,E1 16300.871,E2 16300.871} C_VEL
LIN {X 0,Y 272.203,Z 785.548,A -85,B 0,C 180,E1 16308.591,E2 16308.591} C_VEL
LIN {X 0,Y 277.144,Z 773.254,A -85,B 0,C 180,E1 16315.827,E2 16315.827} C_VEL
LIN {X 0,Y 285.364,Z 754.881,A -85,B 0,C 180,E1 16322.826,E2 16322.826} C_VEL
LIN {X 0,Y 295.461,Z 732.045,A -85,B 0,C 180,E1 16328.735,E2 16328.735} C_VEL
LIN {X 0,Y 306.654,Z 703.993,A -85,B 0,C 180,E1 16333.791,E2 16333.791} C_VEL
LIN {X 0,Y 317.336,Z 672.142,A -85,B 0,C 180,E1 16337.741,E2 16337.741} C_VEL
LIN {X 0,Y 321.702,Z 656.766,A -85,B 0,C 180,E1 16339.154,E2 16339.154} C_VEL
LIN {X 0,Y 316.322,Z 635.845,A -85,B 0,C 180,E1 16343.179,E2 16343.179} C_VEL
LIN {X 0,Y 306.496,Z 612.714,A -85,B 0,C 180,E1 16348.541,E2 16348.541} C_VEL
LIN {X 0,Y 304.127,Z 608.973,A -85,B 0,C 180,E1 16349.716,E2 16349.716} C_VEL
LIN {X 0,Y 296.364,Z 621.854,A -85,B 0,C 180,E1 16350.922,E2 16350.922} C_VEL
LIN {X 0,Y 289.62,Z 633.901,A -85,B 0,C 180,E1 16351.778,E2 16351.778} C_VEL
LIN {X 0,Y 286.187,Z 638.028,A -85,B 0,C 180,E1 16352.48,E2 16352.48} C_VEL
LIN {X 0,Y 280.523,Z 646.797,A -85,B 0,C 180,E1 16353.262,E2 16353.262} C_VEL
LIN {X 0,Y 278.171,Z 647.722,A -85,B 0,C 180,E1 16354.129,E2 16354.129} C_VEL
LIN {X 0,Y 276.941,Z 676.77,A -85,B 0,C 180,E1 16356.298,E2 16356.298} C_VEL
LIN {X 0,Y 275.13,Z 702.836,A -85,B 0,C 180,E1 16359.616,E2 16359.616} C_VEL
LIN {X 0,Y 273.436,Z 723.047,A -85,B 0,C 180,E1 16363.563,E2 16363.563} C_VEL
LIN {X 0,Y 272.376,Z 739.249,A -85,B 0,C 180,E1 16368.407,E2 16368.407} C_VEL
LIN {X 0,Y 272.212,Z 749.618,A -85,B 0,C 180,E1 16373.627,E2 16373.627} C_VEL
LIN {X 0,Y 272.56,Z 753.04,A -85,B 0,C 180,E1 16376.819,E2 16376.819} C_VEL
LIN {X 0,Y 273.368,Z 754.389,A -85,B 0,C 180,E1 16379.993,E2 16379.993} C_VEL
LIN {X 0,Y 275.4,Z 752.516,A -85,B 0,C 180,E1 16384.707,E2 16384.707} C_VEL
LIN {X 0,Y 278.474,Z 745.806,A -85,B 0,C 180,E1 16389.349,E2 16389.349} C_VEL
LIN {X 0,Y 282.533,Z 733.3,A -85,B 0,C 180,E1 16393.9,E2 16393.9} C_VEL
LIN {X 0,Y 287.015,Z 714.797,A -85,B 0,C 180,E1 16397.985,E2 16397.985} C_VEL
LIN {X 0,Y 290.917,Z 692.172,A -85,B 0,C 180,E1 16401.117,E2 16401.117} C_VEL
LIN {X 0,Y 293.569,Z 665.93,A -85,B 0,C 180,E1 16403.369,E2 16403.369} C_VEL
LIN {X 0,Y 296.337,Z 628.688,A -85,B 0,C 180,E1 16405.267,E2 16405.267} C_VEL
LIN {X 0,Y 302.993,Z 617.475,A -85,B 0,C 180,E1 16406.068,E2 16406.068} C_VEL
LIN {X 0,Y 305.983,Z 611.482,A -85,B 0,C 180,E1 16406.343,E2 16406.343} C_VEL
LIN {X 0,Y 317.022,Z 633.945,A -85,B 0,C 180,E1 16412.028,E2 16412.028} C_VEL
LIN {X 0,Y 326.783,Z 661.331,A -85,B 0,C 180,E1 16417.237,E2 16417.237} C_VEL
LIN {X 0,Y 326.676,Z 666.873,A -85,B 0,C 180,E1 16417.842,E2 16417.842} C_VEL
LIN {X 0,Y 315.317,Z 709.678,A -85,B 0,C 180,E1 16421.309,E2 16421.309} C_VEL
LIN {X 0,Y 304.852,Z 741.438,A -85,B 0,C 180,E1 16425.133,E2 16425.133} C_VEL
LIN {X 0,Y 293.747,Z 769.966,A -85,B 0,C 180,E1 16430.032,E2 16430.032} C_VEL
LIN {X 0,Y 283.44,Z 795.084,A -85,B 0,C 180,E1 16436.229,E2 16436.229} C_VEL
LIN {X 0,Y 275.618,Z 814.568,A -85,B 0,C 180,E1 16443.144,E2 16443.144} C_VEL
LIN {X 0,Y 270.875,Z 828.744,A -85,B 0,C 180,E1 16450.47,E2 16450.47} C_VEL
LIN {X 0,Y 268.843,Z 838.666,A -85,B 0,C 180,E1 16458.639,E2 16458.639} C_VEL
LIN {X 0,Y 268.606,Z 843.198,A -85,B 0,C 180,E1 16466.779,E2 16466.779} C_VEL
LIN {X 0,Y 268.992,Z 843.588,A -85,B 0,C 180,E1 16469.999,E2 16469.999} C_VEL
LIN {X 0,Y 268.663,Z 840.766,A -85,B 0,C 180,E1 16478.072,E2 16478.072} C_VEL
LIN {X 0,Y 269.818,Z 832.56,A -85,B 0,C 180,E1 16486.24,E2 16486.24} C_VEL
LIN {X 0,Y 273.593,Z 818.517,A -85,B 0,C 180,E1 16494.351,E2 16494.351} C_VEL
LIN {X 0,Y 280.569,Z 799.009,A -85,B 0,C 180,E1 16501.756,E2 16501.756} C_VEL
LIN {X 0,Y 289.996,Z 774.545,A -85,B 0,C 180,E1 16508.169,E2 16508.169} C_VEL
LIN {X 0,Y 300.654,Z 745.181,A -85,B 0,C 180,E1 16513.512,E2 16513.512} C_VEL
LIN {X 0,Y 310.777,Z 713.286,A -85,B 0,C 180,E1 16517.521,E2 16517.521} C_VEL
LIN {X 0,Y 321.744,Z 670.491,A -85,B 0,C 180,E1 16521.143,E2 16521.143} C_VEL
LIN {X 0,Y 323.342,Z 660.896,A -85,B 0,C 180,E1 16521.904,E2 16521.904} C_VEL
LIN {X 0,Y 322.221,Z 657.078,A -85,B 0,C 180,E1 16522.494,E2 16522.494} C_VEL
LIN {X 0,Y 319.454,Z 657.374,A -85,B 0,C 180,E1 16522.982,E2 16522.982} C_VEL
LIN {X 0,Y 313.514,Z 664.314,A -85,B 0,C 180,E1 16523.345,E2 16523.345} C_VEL
LIN {X 0,Y 302.264,Z 681.375,A -85,B 0,C 180,E1 16523.463,E2 16523.463} C_VEL
LIN {X 0,Y 300.279,Z 683.309,A -85,B 0,C 180,E1 16523.608,E2 16523.608} C_VEL
LIN {X 0,Y 294.723,Z 687.313,A -85,B 0,C 180,E1 16524.389,E2 16524.389} C_VEL
LIN {X 0,Y 288.179,Z 712.213,A -85,B 0,C 180,E1 16527.976,E2 16527.976} C_VEL
LIN {X 0,Y 281.472,Z 731.981,A -85,B 0,C 180,E1 16532.315,E2 16532.315} C_VEL
LIN {X 0,Y 275.19,Z 746.509,A -85,B 0,C 180,E1 16537.435,E2 16537.435} C_VEL
LIN {X 0,Y 270.791,Z 754.116,A -85,B 0,C 180,E1 16542.159,E2 16542.159} C_VEL
LIN {X 0,Y 267.54,Z 757.34,A -85,B 0,C 180,E1 16546.969,E2 16546.969} C_VEL
LIN {X 0,Y 265.968,Z 757.213,A -85,B 0,C 180,E1 16550.207,E2 16550.207} C_VEL
LIN {X 0,Y 264.522,Z 752.833,A -85,B 0,C 180,E1 16555.834,E2 16555.834} C_VEL
LIN {X 0,Y 264.289,Z 743.255,A -85,B 0,C 180,E1 16561.389,E2 16561.389} C_VEL
LIN {X 0,Y 265.204,Z 727.418,A -85,B 0,C 180,E1 16566.952,E2 16566.952} C_VEL
LIN {X 0,Y 266.945,Z 706.606,A -85,B 0,C 180,E1 16571.832,E2 16571.832} C_VEL
LIN {X 0,Y 269.257,Z 681.45,A -85,B 0,C 180,E1 16575.863,E2 16575.863} C_VEL
LIN {X 0,Y 271.419,Z 651.952,A -85,B 0,C 180,E1 16579.004,E2 16579.004} C_VEL
LIN {X 0,Y 272.94,Z 619.216,A -85,B 0,C 180,E1 16581.046,E2 16581.046} C_VEL
LIN {X 0,Y 272.27,Z 601.685,A -85,B 0,C 180,E1 16581.795,E2 16581.795} C_VEL
LIN {X 0,Y 268.995,Z 587.432,A -85,B 0,C 180,E1 16582.739,E2 16582.739} C_VEL
LIN {X 0,Y 271.797,Z 583.666,A -85,B 0,C 180,E1 16583.853,E2 16583.853} C_VEL
LIN {X 0,Y 274.583,Z 578.54,A -85,B 0,C 180,E1 16584.674,E2 16584.674} C_VEL
LIN {X 0,Y 276.326,Z 576.64,A -85,B 0,C 180,E1 16585.371,E2 16585.371} C_VEL
LIN {X 0,Y 285.151,Z 590.66,A -85,B 0,C 180,E1 16591.452,E2 16591.452} C_VEL
LIN {X 0,Y 296.834,Z 612.755,A -85,B 0,C 180,E1 16597.81,E2 16597.81} C_VEL
LIN {X 0,Y 306.113,Z 635.372,A -85,B 0,C 180,E1 16602.683,E2 16602.683} C_VEL
LIN {X 0,Y 311.362,Z 656.495,A -85,B 0,C 180,E1 16606.568,E2 16606.568} C_VEL
LIN {X 0,Y 301.574,Z 689.976,A -85,B 0,C 180,E1 16610.121,E2 16610.121} C_VEL
LIN {X 0,Y 290.83,Z 719.675,A -85,B 0,C 180,E1 16614.74,E2 16614.74} C_VEL
LIN {X 0,Y 280.174,Z 745.673,A -85,B 0,C 180,E1 16620.592,E2 16620.592} C_VEL
LIN {X 0,Y 271.675,Z 765.698,A -85,B 0,C 180,E1 16627.117,E2 16627.117} C_VEL
LIN {X 0,Y 265.411,Z 781.516,A -85,B 0,C 180,E1 16634.876,E2 16634.876} C_VEL
LIN {X 0,Y 262.598,Z 790.295,A -85,B 0,C 180,E1 16641.74,E2 16641.74} C_VEL
LIN {X 0,Y 261.745,Z 794.059,A -85,B 0,C 180,E1 16646.695,E2 16646.695} C_VEL
LIN {X 0,Y 261.305,Z 795.991,A -85,B 0,C 180,E1 16653.312,E2 16653.312} C_VEL
LIN {X 0,Y 262.042,Z 793.34,A -85,B 0,C 180,E1 16661.731,E2 16661.731} C_VEL
LIN {X 0,Y 265.121,Z 785.123,A -85,B 0,C 180,E1 16669.972,E2 16669.972} C_VEL
LIN {X 0,Y 270.757,Z 772.156,A -85,B 0,C 180,E1 16677.378,E2 16677.378} C_VEL
LIN {X 0,Y 279.859,Z 753.004,A -85,B 0,C 180,E1 16684.488,E2 16684.488} C_VEL
LIN {X 0,Y 290.604,Z 729.711,A -85,B 0,C 180,E1 16690.368,E2 16690.368} C_VEL
LIN {X 0,Y 302.272,Z 701.09,A -85,B 0,C 180,E1 16695.356,E2 16695.356} C_VEL
LIN {X 0,Y 313.242,Z 668.666,A -85,B 0,C 180,E1 16699.213,E2 16699.213} C_VEL
LIN {X 0,Y 315.872,Z 658.494,A -85,B 0,C 180,E1 16700.216,E2 16700.216} C_VEL
LIN {X 0,Y 309.409,Z 635.05,A -85,B 0,C 180,E1 16705.12,E2 16705.12} C_VEL
LIN {X 0,Y 302.651,Z 619.671,A -85,B 0,C 180,E1 16709.017,E2 16709.017} C_VEL
LIN {X 0,Y 298.604,Z 625.783,A -85,B 0,C 180,E1 16709.637,E2 16709.637} C_VEL
LIN {X 0,Y 290.856,Z 638.694,A -85,B 0,C 180,E1 16710.559,E2 16710.559} C_VEL
LIN {X 0,Y 287.404,Z 642.877,A -85,B 0,C 180,E1 16711.161,E2 16711.161} C_VEL
LIN {X 0,Y 281.245,Z 651.671,A -85,B 0,C 180,E1 16711.991,E2 16711.991} C_VEL
LIN {X 0,Y 276.322,Z 656.773,A -85,B 0,C 180,E1 16712.994,E2 16712.994} C_VEL
LIN {X 0,Y 272.466,Z 661.332,A -85,B 0,C 180,E1 16713.692,E2 16713.692} C_VEL
LIN {X 0,Y 269.978,Z 662.258,A -85,B 0,C 180,E1 16714.655,E2 16714.655} C_VEL
LIN {X 0,Y 268.429,Z 689.47,A -85,B 0,C 180,E1 16717.349,E2 16717.349} C_VEL
LIN {X 0,Y 266.565,Z 712.798,A -85,B 0,C 180,E1 16720.996,E2 16720.996} C_VEL
LIN {X 0,Y 265.096,Z 731.463,A -85,B 0,C 180,E1 16725.424,E2 16725.424} C_VEL
LIN {X 0,Y 264.382,Z 744.472,A -85,B 0,C 180,E1 16730.133,E2 16730.133} C_VEL
LIN {X 0,Y 264.57,Z 753.181,A -85,B 0,C 180,E1 16735.639,E2 16735.639} C_VEL
LIN {X 0,Y 265.584,Z 755.824,A -85,B 0,C 180,E1 16739.993,E2 16739.993} C_VEL
LIN {X 0,Y 267.753,Z 754.44,A -85,B 0,C 180,E1 16744.842,E2 16744.842} C_VEL
LIN {X 0,Y 271.022,Z 748.194,A -85,B 0,C 180,E1 16749.608,E2 16749.608} C_VEL
LIN {X 0,Y 275.335,Z 736.401,A -85,B 0,C 180,E1 16754.271,E2 16754.271} C_VEL
LIN {X 0,Y 280.157,Z 718.862,A -85,B 0,C 180,E1 16758.441,E2 16758.441} C_VEL
LIN {X 0,Y 284.536,Z 696.627,A -85,B 0,C 180,E1 16761.785,E2 16761.785} C_VEL
LIN {X 0,Y 287.757,Z 669.663,A -85,B 0,C 180,E1 16764.281,E2 16764.281} C_VEL
LIN {X 0,Y 289.828,Z 646.669,A -85,B 0,C 180,E1 16765.638,E2 16765.638} C_VEL
LIN {X 0,Y 296.436,Z 636.53,A -85,B 0,C 180,E1 16766.415,E2 16766.415} C_VEL
LIN {X 0,Y 304.623,Z 622.75,A -85,B 0,C 180,E1 16767.253,E2 16767.253} C_VEL
LIN {X 0,Y 313.87,Z 643.516,A -85,B 0,C 180,E1 16772.328,E2 16772.328} C_VEL
LIN {X 0,Y 321.328,Z 666.078,A -85,B 0,C 180,E1 16776.683,E2 16776.683} C_VEL
LIN {X 0,Y 309.451,Z 710.41,A -85,B 0,C 180,E1 16780.356,E2 16780.356} C_VEL
LIN {X 0,Y 298.195,Z 742.903,A -85,B 0,C 180,E1 16784.366,E2 16784.366} C_VEL
LIN {X 0,Y 286.67,Z 771.064,A -85,B 0,C 180,E1 16789.377,E2 16789.377} C_VEL
LIN {X 0,Y 276.097,Z 795.416,A -85,B 0,C 180,E1 16795.63,E2 16795.63} C_VEL
LIN {X 0,Y 267.565,Z 815.636,A -85,B 0,C 180,E1 16803.177,E2 16803.177} C_VEL
LIN {X 0,Y 262.744,Z 829.658,A -85,B 0,C 180,E1 16810.998,E2 16810.998} C_VEL
LIN {X 0,Y 260.88,Z 838.954,A -85,B 0,C 180,E1 16819.486,E2 16819.486} C_VEL
LIN {X 0,Y 260.714,Z 842.494,A -85,B 0,C 180,E1 16826.681,E2 16826.681} C_VEL
LIN {X 0,Y 261.135,Z 842.88,A -85,B 0,C 180,E1 16829.999,E2 16829.999} C_VEL
LIN {X 0,Y 260.788,Z 840.019,A -85,B 0,C 180,E1 16838.318,E2 16838.318} C_VEL
LIN {X 0,Y 262.077,Z 831.748,A -85,B 0,C 180,E1 16846.733,E2 16846.733} C_VEL
LIN {X 0,Y 265.904,Z 818.223,A -85,B 0,C 180,E1 16854.785,E2 16854.785} C_VEL
LIN {X 0,Y 273.439,Z 798.345,A -85,B 0,C 180,E1 16862.556,E2 16862.556} C_VEL
LIN {X 0,Y 283.526,Z 773.38,A -85,B 0,C 180,E1 16869.204,E2 16869.204} C_VEL
LIN {X 0,Y 294.512,Z 744.369,A -85,B 0,C 180,E1 16874.538,E2 16874.538} C_VEL
LIN {X 0,Y 305.27,Z 711.594,A -85,B 0,C 180,E1 16878.662,E2 16878.662} C_VEL
LIN {X 0,Y 315.962,Z 670.59,A -85,B 0,C 180,E1 16882.17,E2 16882.17} C_VEL
LIN {X 0,Y 300.279,Z 683.309,A -85,B 0,C 180,E1 16883.608,E2 16883.608} C_VEL
LIN {X 0,Y 288.687,Z 697.632,A -85,B 0,C 180,E1 16884.358,E2 16884.358} C_VEL
LIN {X 0,Y 286.921,Z 701.882,A -85,B 0,C 180,E1 16884.815,E2 16884.815} C_VEL
LIN {X 0,Y 279.037,Z 725.385,A -85,B 0,C 180,E1 16889.094,E2 16889.094} C_VEL
LIN {X 0,Y 271.69,Z 742.582,A -85,B 0,C 180,E1 16894.07,E2 16894.07} C_VEL
LIN {X 0,Y 265.718,Z 753.144,A -85,B 0,C 180,E1 16899.218,E2 16899.218} C_VEL
LIN {X 0,Y 262.257,Z 757.572,A -85,B 0,C 180,E1 16903.288,E2 16903.288} C_VEL
LIN {X 0,Y 260.023,Z 759.079,A -85,B 0,C 180,E1 16906.585,E2 16906.585} C_VEL
LIN {X 0,Y 257.719,Z 757.937,A -85,B 0,C 180,E1 16911.59,E2 16911.59} C_VEL
LIN {X 0,Y 256.538,Z 751.573,A -85,B 0,C 180,E1 16917.479,E2 16917.479} C_VEL
LIN {X 0,Y 256.663,Z 739.381,A -85,B 0,C 180,E1 16923.378,E2 16923.378} C_VEL
LIN {X 0,Y 257.846,Z 721.599,A -85,B 0,C 180,E1 16928.845,E2 16928.845} C_VEL
LIN {X 0,Y 259.988,Z 698.58,A -85,B 0,C 180,E1 16933.646,E2 16933.646} C_VEL
LIN {X 0,Y 262.43,Z 670.924,A -85,B 0,C 180,E1 16937.544,E2 16937.544} C_VEL
LIN {X 0,Y 264.493,Z 639.105,A -85,B 0,C 180,E1 16940.378,E2 16940.378} C_VEL
LIN {X 0,Y 265.018,Z 604.477,A -85,B 0,C 180,E1 16942.101,E2 16942.101} C_VEL
LIN {X 0,Y 264.299,Z 601.185,A -85,B 0,C 180,E1 16942.337,E2 16942.337} C_VEL
LIN {X 0,Y 266.715,Z 598.59,A -85,B 0,C 180,E1 16943.415,E2 16943.415} C_VEL
LIN {X 0,Y 269.873,Z 592.774,A -85,B 0,C 180,E1 16944.32,E2 16944.32} C_VEL
LIN {X 0,Y 274.068,Z 585.448,A -85,B 0,C 180,E1 16945.504,E2 16945.504} C_VEL
LIN {X 0,Y 275.696,Z 587.264,A -85,B 0,C 180,E1 16946.685,E2 16946.685} C_VEL
LIN {X 0,Y 284.737,Z 602.808,A -85,B 0,C 180,E1 16952.765,E2 16952.765} C_VEL
LIN {X 0,Y 296.181,Z 626.631,A -85,B 0,C 180,E1 16959.097,E2 16959.097} C_VEL
LIN {X 0,Y 303.33,Z 648.805,A -85,B 0,C 180,E1 16963.716,E2 16963.716} C_VEL
LIN {X 0,Y 305.287,Z 659.54,A -85,B 0,C 180,E1 16965.713,E2 16965.713} C_VEL
LIN {X 0,Y 295.183,Z 692.418,A -85,B 0,C 180,E1 16969.319,E2 16969.319} C_VEL
LIN {X 0,Y 284.458,Z 720.731,A -85,B 0,C 180,E1 16973.827,E2 16973.827} C_VEL
LIN {X 0,Y 273.768,Z 745.75,A -85,B 0,C 180,E1 16979.542,E2 16979.542} C_VEL
LIN {X 0,Y 264.435,Z 766.583,A -85,B 0,C 180,E1 16986.454,E2 16986.454} C_VEL
LIN {X 0,Y 258.062,Z 781.664,A -85,B 0,C 180,E1 16994.012,E2 16994.012} C_VEL
LIN {X 0,Y 254.831,Z 791.063,A -85,B 0,C 180,E1 17001.486,E2 17001.486} C_VEL
LIN {X 0,Y 253.908,Z 794.794,A -85,B 0,C 180,E1 17006.593,E2 17006.593} C_VEL
LIN {X 0,Y 253.453,Z 796.702,A -85,B 0,C 180,E1 17013.414,E2 17013.414} C_VEL
LIN {X 0,Y 254.264,Z 794.021,A -85,B 0,C 180,E1 17022.095,E2 17022.095} C_VEL
LIN {X 0,Y 257.62,Z 785.778,A -85,B 0,C 180,E1 17030.579,E2 17030.579} C_VEL
LIN {X 0,Y 263.654,Z 772.8,A -85,B 0,C 180,E1 17038.18,E2 17038.18} C_VEL
LIN {X 0,Y 273.277,Z 753.643,A -85,B 0,C 180,E1 17045.442,E2 17045.442} C_VEL
LIN {X 0,Y 284.83,Z 729.598,A -85,B 0,C 180,E1 17051.571,E2 17051.571} C_VEL
LIN {X 0,Y 296.737,Z 701.679,A -85,B 0,C 180,E1 17056.449,E2 17056.449} C_VEL
LIN {X 0,Y 307.799,Z 670.305,A -85,B 0,C 180,E1 17060.222,E2 17060.222} C_VEL
LIN {X 0,Y 310.072,Z 661.47,A -85,B 0,C 180,E1 17061.147,E2 17061.147} C_VEL
LIN {X 0,Y 303.73,Z 637.646,A -85,B 0,C 180,E1 17066.416,E2 17066.416} C_VEL
LIN {X 0,Y 300.995,Z 630.279,A -85,B 0,C 180,E1 17068.257,E2 17068.257} C_VEL
LIN {X 0,Y 290.643,Z 645.036,A -85,B 0,C 180,E1 17069.58,E2 17069.58} C_VEL
LIN {X 0,Y 281.321,Z 657.117,A -85,B 0,C 180,E1 17070.831,E2 17070.831} C_VEL
LIN {X 0,Y 270.614,Z 667.894,A -85,B 0,C 180,E1 17072.86,E2 17072.86} C_VEL
LIN {X 0,Y 267.429,Z 670.713,A -85,B 0,C 180,E1 17073.609,E2 17073.609} C_VEL
LIN {X 0,Y 263.307,Z 674.55,A -85,B 0,C 180,E1 17074.535,E2 17074.535} C_VEL
LIN {X 0,Y 261.632,Z 675.313,A -85,B 0,C 180,E1 17075.387,E2 17075.387} C_VEL
LIN {X 0,Y 259.809,Z 701.398,A -85,B 0,C 180,E1 17078.656,E2 17078.656} C_VEL
LIN {X 0,Y 257.888,Z 723.642,A -85,B 0,C 180,E1 17082.98,E2 17082.98} C_VEL
LIN {X 0,Y 256.737,Z 740.734,A -85,B 0,C 180,E1 17088.12,E2 17088.12} C_VEL
LIN {X 0,Y 256.534,Z 751.165,A -85,B 0,C 180,E1 17093.236,E2 17093.236} C_VEL
LIN {X 0,Y 256.977,Z 755.345,A -85,B 0,C 180,E1 17096.749,E2 17096.749} C_VEL
LIN {X 0,Y 257.801,Z 757.203,A -85,B 0,C 180,E1 17099.992,E2 17099.992} C_VEL
LIN {X 0,Y 260.109,Z 756.296,A -85,B 0,C 180,E1 17104.985,E2 17104.985} C_VEL
LIN {X 0,Y 263.577,Z 750.662,A -85,B 0,C 180,E1 17109.882,E2 17109.882} C_VEL
LIN {X 0,Y 268.618,Z 738.33,A -85,B 0,C 180,E1 17115.052,E2 17115.052} C_VEL
LIN {X 0,Y 274.178,Z 719.72,A -85,B 0,C 180,E1 17119.562,E2 17119.562} C_VEL
LIN {X 0,Y 278.964,Z 697.403,A -85,B 0,C 180,E1 17122.935,E2 17122.935} C_VEL
LIN {X 0,Y 282.451,Z 670.264,A -85,B 0,C 180,E1 17125.461,E2 17125.461} C_VEL
LIN {X 0,Y 283.525,Z 662.492,A -85,B 0,C 180,E1 17126.019,E2 17126.019} C_VEL
LIN {X 0,Y 289.806,Z 654.028,A -85,B 0,C 180,E1 17126.793,E2 17126.793} C_VEL
LIN {X 0,Y 299.75,Z 638.443,A -85,B 0,C 180,E1 17127.746,E2 17127.746} C_VEL
LIN {X 0,Y 303.1,Z 634.2,A -85,B 0,C 180,E1 17128.22,E2 17128.22} C_VEL
LIN {X 0,Y 311.799,Z 656.901,A -85,B 0,C 180,E1 17133.439,E2 17133.439} C_VEL
LIN {X 0,Y 315.311,Z 670.612,A -85,B 0,C 180,E1 17135.956,E2 17135.956} C_VEL
LIN {X 0,Y 303.184,Z 712.555,A -85,B 0,C 180,E1 17139.506,E2 17139.506} C_VEL
LIN {X 0,Y 291.599,Z 744.28,A -85,B 0,C 180,E1 17143.566,E2 17143.566} C_VEL
LIN {X 0,Y 279.734,Z 771.79,A -85,B 0,C 180,E1 17148.631,E2 17148.631} C_VEL
LIN {X 0,Y 268.483,Z 796.433,A -85,B 0,C 180,E1 17155.222,E2 17155.222} C_VEL
LIN {X 0,Y 259.835,Z 815.959,A -85,B 0,C 180,E1 17162.859,E2 17162.859} C_VEL
LIN {X 0,Y 254.672,Z 830.318,A -85,B 0,C 180,E1 17171.428,E2 17171.428} C_VEL
LIN {X 0,Y 252.982,Z 838.612,A -85,B 0,C 180,E1 17179.69,E2 17179.69} C_VEL
LIN {X 0,Y 252.821,Z 841.791,A -85,B 0,C 180,E1 17186.577,E2 17186.577} C_VEL
LIN {X 0,Y 253.258,Z 842.17,A -85,B 0,C 180,E1 17189.999,E2 17189.999} C_VEL
LIN {X 0,Y 252.905,Z 839.269,A -85,B 0,C 180,E1 17198.579,E2 17198.579} C_VEL
LIN {X 0,Y 254.319,Z 830.929,A -85,B 0,C 180,E1 17207.259,E2 17207.259} C_VEL
LIN {X 0,Y 258.462,Z 817.314,A -85,B 0,C 180,E1 17215.55,E2 17215.55} C_VEL
LIN {X 0,Y 266.522,Z 797.325,A -85,B 0,C 180,E1 17223.51,E2 17223.51} C_VEL
LIN {X 0,Y 276.929,Z 772.651,A -85,B 0,C 180,E1 17230.189,E2 17230.189} C_VEL
LIN {X 0,Y 288.449,Z 743.646,A -85,B 0,C 180,E1 17235.59,E2 17235.59} C_VEL
LIN {X 0,Y 299.384,Z 711.535,A -85,B 0,C 180,E1 17239.679,E2 17239.679} C_VEL
LIN {X 0,Y 306.481,Z 686.38,A -85,B 0,C 180,E1 17241.987,E2 17241.987} C_VEL
LIN {X 0,Y 305.366,Z 685.954,A -85,B 0,C 180,E1 17242.255,E2 17242.255} C_VEL
LIN {X 0,Y 288.921,Z 696.91,A -85,B 0,C 180,E1 17244.023,E2 17244.023} C_VEL
LIN {X 0,Y 286.921,Z 701.882,A -85,B 0,C 180,E1 17244.815,E2 17244.815} C_VEL
LIN {X 0,Y 281.774,Z 711.844,A -85,B 0,C 180,E1 17245.623,E2 17245.623} C_VEL
LIN {X 0,Y 276.293,Z 721.227,A -85,B 0,C 180,E1 17246.569,E2 17246.569} C_VEL
LIN {X 0,Y 267.93,Z 740.005,A -85,B 0,C 180,E1 17251.412,E2 17251.412} C_VEL
LIN {X 0,Y 260.44,Z 752.981,A -85,B 0,C 180,E1 17256.985,E2 17256.985} C_VEL
LIN {X 0,Y 254.927,Z 759.563,A -85,B 0,C 180,E1 17262.792,E2 17262.792} C_VEL
LIN {X 0,Y 252.521,Z 760.801,A -85,B 0,C 180,E1 17266.179,E2 17266.179} C_VEL
